(* IEC 61131-3 sources: SRCI/RobotLibrary/Library/POUs/AdvancedMove/MC_MoveLinearOffset, 1 file *)

(* ---- MC_MoveLinearOffsetFB.st ---- *)
/// Move the TCP relative to a reference cartesian position (linear interpolation)
FUNCTION_BLOCK MC_MoveLinearOffsetFB EXTENDS RobotLibraryBaseExecuteFB
// -------------------------------------------------------------------------
//  SRCI Robot Library
// -------------------------------------------------------------------------
//
//  Object:      MoveLinearOffsetFB
//  Author:      Thorsten Brach
//  Date:        2024-06-01
//
//  Description:
//
//
//  Copyright:
//    (C) 2024 Thorsten Brach. All rights reserved
//             Licensed under the LGPL-3.0 license.
//
//  Disclaimer:
//    This project is provided without any guarantee and can be used for
//    private and commercial purposes. Any use is at the user’s
//    own risk and responsibility.
//
// -------------------------------------------------------------------------
VAR_INPUT
  /// Parameter which determines the behavior towards the previously sent and still active or buffered commands
  AbortingMode       : AbortingMode;
  /// Defines the target sequence in which the command will be executed
  SequenceFlag       : SequenceFlag;
  /// command parameter
  ParCmd             : MoveLinearOffsetParCmd;
END_VAR

VAR_OUTPUT
  /// Command is transferred and confirmed by the RC
  CommandBuffered    : BOOL;
  /// The command takes control of the motion of the according axis group
  Active             : BOOL;
  /// The command was aborted by another command.
  CommandAborted     : BOOL;
  /// TRUE, while command is interrupted during execution and can be continued
  CommandInterrupted : BOOL;
  /// command outputs
  OutCmd             : MoveLinearOffsetOutCmd;
END_VAR

VAR
  /// internal copy of command parameter
 _parCmd             : MoveLinearOffsetParCmd;
  /// command data to send
 _command            : MoveLinearOffsetSendData;
  /// response data received
 _response           : MoveLinearOffsetRecvData;
END_VAR

  SUPER^(AxesGroup := AxesGroup);

END_FUNCTION_BLOCK

METHOD INTERNAL CheckAddParameter : BOOL
VAR_INPUT
  /// Payload pointer
  PayloadPtr : UDINT;
END_VAR
VAR
  /// Payload as byte array
  Payload    : ARRAY [1..SIZEOF(_command)] OF BYTE;
  /// Null Byte array
  Null       : ARRAY [1..SIZEOF(_command)] OF BYTE;
  /// Data length to compare
  DataLen    : UDINT;
END_VAR

  // Payload pointer must be decreased by one byte, because ADR(Payload) is already one byte !
  PayloadPtr := LIMIT (0, PayloadPtr - 1, SIZEOF(Payload) -1);
  // Convert command struct to payload array
  SysDepMemCpy( pDest := ADR(Payload), pSrc := ADR(_command), DataLen := SIZEOF(_command));
  // Calculate the data length to compare - at least one byte must be compared !
  DataLen := LIMIT(1, SIZEOF(Payload) - PayloadPtr, SIZEOF(Payload));
  // Compare Payload-Array with Null-Byte-Array
  CheckAddParameter := SysDepMemCmp( pData1 := ADR(Payload) + PayloadPtr , pData2 := ADR(Null), DataLen := DataLen) <>  RobotLibraryConstants.OK ;

END_METHOD

METHOD PROTECTED CheckFunctionSupported : BOOL
VAR_IN_OUT
  /// Robot assignment of function
  AxesGroup : AxesGroup;
END_VAR

  CheckFunctionSupported := AxesGroup.State.RobotData.RCSupportedFunctions.MoveLinearOffset;

  IF ( NOT CheckFunctionSupported )
  THEN
    // call base implementation for set error and create log entry
    SUPER^.CheckFunctionSupported(AxesGroup := AxesGroup);
  END_IF

END_METHOD

METHOD PROTECTED CheckParameterChanged : BOOL
VAR_IN_OUT
  /// Robot assignment of function
  AxesGroup    : AxesGroup;
END_VAR

  // Check ParCmd Size is > 0, because MemCmp does not work correctly with size = 0
  IF (SIZEOF(ParCmd) = 0) OR (_stepCmd = 0)
  THEN
    RETURN;
  END_IF

  // compare memory
  _parameterChanged := ( SysDepMemCmp(pData1 := ADR(ParCmd), pData2 := ADR(_parCmd), DataLen := SIZEOF(ParCmd)) <> RobotLibraryConstants.OK );

  // check parameter valid ?
  _parameterValid   := CheckParameterValid( AxesGroup := AxesGroup );

  IF ((  _parameterChanged        )  AND
      (  _parameterValid          )) OR
      (  _parameterUpdateInternal )
  THEN
    // reset internal flag for send parameter update
   _parameterUpdateInternal := FALSE;
    // update internal copy of parameters
   _parCmd := ParCmd;
    // inc parameter sequence
   _command.ParSeq := _command.ParSeq + 1;
    // update command data
    CommandData := CreateCommandPayload(AxesGroup := AxesGroup); // ( Access via reference to rCommandFB in ACR )
    // notify active command register
    AxesGroup.Acyclic.ActiveCommandRegister.NotifyParameterChanged := _uniqueID;
  END_IF

END_METHOD

METHOD PROTECTED CheckParameterValid : BOOL
VAR_IN_OUT
  /// Robot assignment of function
  AxesGroup : AxesGroup;
END_VAR
VAR
  /// internal index for loops
 _idx : DINT;
END_VAR

  CheckParameterValid := TRUE;

  // Check AbortingMode valid ?
  IF (( AbortingMode <> AbortingModeEnum.BUFFER ) AND
      ( AbortingMode <> AbortingModeEnum.ABORT  ))
  THEN
    // Parameter not valid
    CheckParameterValid := FALSE;
    // Set error
    ErrorID := RobotLibraryErrorIdEnum.ERR_ABORTINGMODE_INVALID;
    // Create log entry
    CreateLogMessagePara1 ( Timestamp   := AxesGroup.State.SystemTime,
                            MessageType := MessageType.CMD,
                            Severity    := Severity.ERROR,
                            MessageCode := ErrorID,
                            MessageText := 'Invalid Parameter AbortingMode = {1}',
                            Para1       := ABORTING_MODE_TO_STRING(AbortingMode));
    RETURN;
  END_IF

  // Check SequenceFlag valid ?
  IF (( SequenceFlag <> SequenceFlagEnum.PRIMARY_SEQUENCE   ) AND
      ( SequenceFlag <> SequenceFlagEnum.SECONDARY_SEQUENCE ))
  THEN
    // Parameter not valid
    CheckParameterValid := FALSE;
    // Set error
    ErrorID := RobotLibraryErrorIdEnum.ERR_SEQFLAG_NOT_ALLOWED;
    // Create log entry
    CreateLogMessagePara1 ( Timestamp   := AxesGroup.State.SystemTime,
                            MessageType := MessageType.CMD,
                            Severity    := Severity.ERROR,
                            MessageCode := ErrorID,
                            MessageText := 'Invalid Parameter SequenceFlag = {1}',
                            Para1       := SEQUENCE_FLAG_TO_STRING(SequenceFlag));
    RETURN;
  END_IF

  // Check ParCmd.ReferencePosition.X valid ?
  IF ( SysDepIsValidReal(ParCmd.ReferencePosition.X) = FALSE )
  THEN
    // Parameter not valid
    CheckParameterValid := FALSE;
    // Set error
    ErrorID := RobotLibraryErrorIdEnum.ERR_INVALID_PAR_CMD;

    // Create log entry
    CreateLogMessagePara1 ( Timestamp   := AxesGroup.State.SystemTime,
                            MessageType := MessageType.CMD,
                            Severity    := Severity.ERROR,
                            MessageCode := ErrorID,
                            MessageText := 'Invalid Parameter ParCmd.ReferencePosition.X = {1}',
                            Para1       := VALID_REAL_TO_STRING(ParCmd.ReferencePosition.X));
    RETURN;
  END_IF

  // Check ParCmd.ReferencePosition.Y valid ?
  IF ( SysDepIsValidReal(ParCmd.ReferencePosition.Y) = FALSE )
  THEN
    // Parameter not valid
    CheckParameterValid := FALSE;
    // Set error
    ErrorID := RobotLibraryErrorIdEnum.ERR_INVALID_PAR_CMD;

    // Create log entry
    CreateLogMessagePara1 ( Timestamp   := AxesGroup.State.SystemTime,
                            MessageType := MessageType.CMD,
                            Severity    := Severity.ERROR,
                            MessageCode := ErrorID,
                            MessageText := 'Invalid Parameter ParCmd.ReferencePosition.Y = {1}',
                            Para1       := VALID_REAL_TO_STRING(ParCmd.ReferencePosition.Y));
    RETURN;
  END_IF

  // Check ParCmd.ReferencePosition.Z valid ?
  IF ( SysDepIsValidReal(ParCmd.ReferencePosition.Z) = FALSE )
  THEN
    // Parameter not valid
    CheckParameterValid := FALSE;
    // Set error
    ErrorID := RobotLibraryErrorIdEnum.ERR_INVALID_PAR_CMD;

    // Create log entry
    CreateLogMessagePara1 ( Timestamp   := AxesGroup.State.SystemTime,
                            MessageType := MessageType.CMD,
                            Severity    := Severity.ERROR,
                            MessageCode := ErrorID,
                            MessageText := 'Invalid Parameter ParCmd.ReferencePosition.Z = {1}',
                            Para1       := VALID_REAL_TO_STRING(ParCmd.ReferencePosition.Z));
    RETURN;
  END_IF

  // Check ParCmd.ReferencePosition.Rx valid ?
  IF ( SysDepIsValidReal(ParCmd.ReferencePosition.Rx) = FALSE )
  THEN
    // Parameter not valid
    CheckParameterValid := FALSE;
    // Set error
    ErrorID := RobotLibraryErrorIdEnum.ERR_INVALID_PAR_CMD;

    // Create log entry
    CreateLogMessagePara1 ( Timestamp   := AxesGroup.State.SystemTime,
                            MessageType := MessageType.CMD,
                            Severity    := Severity.ERROR,
                            MessageCode := ErrorID,
                            MessageText := 'Invalid Parameter ParCmd.ReferencePosition.Rx = {1}',
                            Para1       := VALID_REAL_TO_STRING(ParCmd.ReferencePosition.Rx));
    RETURN;
  END_IF

  // Check ParCmd.ReferencePosition.Ry valid ?
  IF ( SysDepIsValidReal(ParCmd.ReferencePosition.Ry) = FALSE )
  THEN
    // Parameter not valid
    CheckParameterValid := FALSE;
    // Set error
    ErrorID := RobotLibraryErrorIdEnum.ERR_INVALID_PAR_CMD;

    // Create log entry
    CreateLogMessagePara1 ( Timestamp   := AxesGroup.State.SystemTime,
                            MessageType := MessageType.CMD,
                            Severity    := Severity.ERROR,
                            MessageCode := ErrorID,
                            MessageText := 'Invalid Parameter ParCmd.ReferencePosition.Ry = {1}',
                            Para1       := VALID_REAL_TO_STRING(ParCmd.ReferencePosition.Ry));
    RETURN;
  END_IF

  // Check ParCmd.ReferencePosition.Rz valid ?
  IF ( SysDepIsValidReal(ParCmd.ReferencePosition.Rz) = FALSE )
  THEN
    // Parameter not valid
    CheckParameterValid := FALSE;
    // Set error
    ErrorID := RobotLibraryErrorIdEnum.ERR_INVALID_PAR_CMD;

    // Create log entry
    CreateLogMessagePara1 ( Timestamp   := AxesGroup.State.SystemTime,
                            MessageType := MessageType.CMD,
                            Severity    := Severity.ERROR,
                            MessageCode := ErrorID,
                            MessageText := 'Invalid Parameter ParCmd.ReferencePosition.Rz = {1}',
                            Para1       := VALID_REAL_TO_STRING(ParCmd.ReferencePosition.Rz));
    RETURN;
  END_IF

  // Check ParCmd.ReferencePosition.E1 valid ?
  IF ( SysDepIsValidReal(ParCmd.ReferencePosition.E1) = FALSE )
  THEN
    // Parameter not valid
    CheckParameterValid := FALSE;
    // Set error
    ErrorID := RobotLibraryErrorIdEnum.ERR_INVALID_PAR_CMD;

    // Create log entry
    CreateLogMessagePara1 ( Timestamp   := AxesGroup.State.SystemTime,
                            MessageType := MessageType.CMD,
                            Severity    := Severity.ERROR,
                            MessageCode := ErrorID,
                            MessageText := 'Invalid Parameter ParCmd.ReferencePosition.E1 = {1}',
                            Para1       := VALID_REAL_TO_STRING(ParCmd.ReferencePosition.E1));
    RETURN;
  END_IF

  // Check ParCmd.ReferencePosition.E2 valid ?
  IF ( SysDepIsValidReal(ParCmd.ReferencePosition.E2) = FALSE )
  THEN
    // Parameter not valid
    CheckParameterValid := FALSE;
    // Set error
    ErrorID := RobotLibraryErrorIdEnum.ERR_INVALID_PAR_CMD;

    // Create log entry
    CreateLogMessagePara1 ( Timestamp   := AxesGroup.State.SystemTime,
                            MessageType := MessageType.CMD,
                            Severity    := Severity.ERROR,
                            MessageCode := ErrorID,
                            MessageText := 'Invalid Parameter ParCmd.ReferencePosition.E2 = {1}',
                            Para1       := VALID_REAL_TO_STRING(ParCmd.ReferencePosition.E2));
    RETURN;
  END_IF

  // Check ParCmd.ReferencePosition.E3 valid ?
  IF ( SysDepIsValidReal(ParCmd.ReferencePosition.E3) = FALSE )
  THEN
    // Parameter not valid
    CheckParameterValid := FALSE;
    // Set error
    ErrorID := RobotLibraryErrorIdEnum.ERR_INVALID_PAR_CMD;

    // Create log entry
    CreateLogMessagePara1 ( Timestamp   := AxesGroup.State.SystemTime,
                            MessageType := MessageType.CMD,
                            Severity    := Severity.ERROR,
                            MessageCode := ErrorID,
                            MessageText := 'Invalid Parameter ParCmd.ReferencePosition.E3 = {1}',
                            Para1       := VALID_REAL_TO_STRING(ParCmd.ReferencePosition.E3));
    RETURN;
  END_IF

  // Check ParCmd.ReferencePosition.E4 valid ?
  IF ( SysDepIsValidReal(ParCmd.ReferencePosition.E4) = FALSE )
  THEN
    // Parameter not valid
    CheckParameterValid := FALSE;
    // Set error
    ErrorID := RobotLibraryErrorIdEnum.ERR_INVALID_PAR_CMD;

    // Create log entry
    CreateLogMessagePara1 ( Timestamp   := AxesGroup.State.SystemTime,
                            MessageType := MessageType.CMD,
                            Severity    := Severity.ERROR,
                            MessageCode := ErrorID,
                            MessageText := 'Invalid Parameter ParCmd.ReferencePosition.E4 = {1}',
                            Para1       := VALID_REAL_TO_STRING(ParCmd.ReferencePosition.E4));
    RETURN;
  END_IF

  // Check ParCmd.ReferencePosition.E5 valid ?
  IF ( SysDepIsValidReal(ParCmd.ReferencePosition.E5) = FALSE )
  THEN
    // Parameter not valid
    CheckParameterValid := FALSE;
    // Set error
    ErrorID := RobotLibraryErrorIdEnum.ERR_INVALID_PAR_CMD;

    // Create log entry
    CreateLogMessagePara1 ( Timestamp   := AxesGroup.State.SystemTime,
                            MessageType := MessageType.CMD,
                            Severity    := Severity.ERROR,
                            MessageCode := ErrorID,
                            MessageText := 'Invalid Parameter ParCmd.ReferencePosition.E5 = {1}',
                            Para1       := VALID_REAL_TO_STRING(ParCmd.ReferencePosition.E5));
    RETURN;
  END_IF

  // Check ParCmd.ReferencePosition.E6 valid ?
  IF ( SysDepIsValidReal(ParCmd.ReferencePosition.E6) = FALSE )
  THEN
    // Parameter not valid
    CheckParameterValid := FALSE;
    // Set error
    ErrorID := RobotLibraryErrorIdEnum.ERR_INVALID_PAR_CMD;

    // Create log entry
    CreateLogMessagePara1 ( Timestamp   := AxesGroup.State.SystemTime,
                            MessageType := MessageType.CMD,
                            Severity    := Severity.ERROR,
                            MessageCode := ErrorID,
                            MessageText := 'Invalid Parameter ParCmd.ReferencePosition.E6 = {1}',
                            Para1       := VALID_REAL_TO_STRING(ParCmd.ReferencePosition.E6));
    RETURN;
  END_IF

  // Check ParCmd.ReferencePosition.Config.Shoulder valid ?
  IF (( ParCmd.ReferencePosition.Config.Shoulder <> ArmConfigShoulder.USE_CONFIG ) AND
      ( ParCmd.ReferencePosition.Config.Shoulder <> ArmConfigShoulder.SAME       ) AND
      ( ParCmd.ReferencePosition.Config.Shoulder <> ArmConfigShoulder.FREE       ) AND
      ( ParCmd.ReferencePosition.Config.Shoulder <> ArmConfigShoulder.BACK       ) AND
      ( ParCmd.ReferencePosition.Config.Shoulder <> ArmConfigShoulder.FRONT      ))
  THEN
    // Parameter not valid
    CheckParameterValid := FALSE;
    // Set error
    ErrorID := RobotLibraryErrorIdEnum.ERR_CONFIGMODE_SHOULDER_INVALID;
    // Create log entry
    CreateLogMessagePara1 ( Timestamp   := AxesGroup.State.SystemTime,
                            MessageType := MessageType.CMD,
                            Severity    := Severity.ERROR,
                            MessageCode := ErrorID,
                            MessageText := 'Invalid Parameter ParCmd.ReferencePosition.Config.Shoulder = {1}',
                            Para1       :=  ARM_CONFIG_SHOULDER_TO_STRING(ParCmd.ReferencePosition.Config.Shoulder));
    RETURN;
  END_IF

  // Check ParCmd.ReferencePosition.Config.Elbow valid ?
  IF (( ParCmd.ReferencePosition.Config.Elbow <> ArmConfigElbow.USE_CONFIG ) AND
      ( ParCmd.ReferencePosition.Config.Elbow <> ArmConfigElbow.SAME       ) AND
      ( ParCmd.ReferencePosition.Config.Elbow <> ArmConfigElbow.FREE       ) AND
      ( ParCmd.ReferencePosition.Config.Elbow <> ArmConfigElbow.DOWN       ) AND
      ( ParCmd.ReferencePosition.Config.Elbow <> ArmConfigElbow.UP         ))
  THEN
    // Parameter not valid
    CheckParameterValid := FALSE;
    // Set error
    ErrorID := RobotLibraryErrorIdEnum.ERR_CONFIGMODE_ELBOW_INVALID;
    // Create log entry
    CreateLogMessagePara1 ( Timestamp   := AxesGroup.State.SystemTime,
                            MessageType := MessageType.CMD,
                            Severity    := Severity.ERROR,
                            MessageCode := ErrorID,
                            MessageText := 'Invalid Parameter ParCmd.ReferencePosition.Config.Elbow = {1}',
                            Para1       :=  ARM_CONFIG_ELBOW_TO_STRING(ParCmd.ReferencePosition.Config.Elbow));
    RETURN;
  END_IF

  // Check ParCmd.ReferencePosition.Config.Wrist valid ?
  IF (( ParCmd.ReferencePosition.Config.Wrist <> ArmConfigWrist.USE_CONFIG ) AND
      ( ParCmd.ReferencePosition.Config.Wrist <> ArmConfigWrist.SAME       ) AND
      ( ParCmd.ReferencePosition.Config.Wrist <> ArmConfigWrist.FREE       ) AND
      ( ParCmd.ReferencePosition.Config.Wrist <> ArmConfigWrist.FLIP       ) AND
      ( ParCmd.ReferencePosition.Config.Wrist <> ArmConfigWrist.NON_FLIP   ))
  THEN
    // Parameter not valid
    CheckParameterValid := FALSE;
    // Set error
    ErrorID := RobotLibraryErrorIdEnum.ERR_CONFIGMODE_WRIST_INVALID;
    // Create log entry
    CreateLogMessagePara1 ( Timestamp   := AxesGroup.State.SystemTime,
                            MessageType := MessageType.CMD,
                            Severity    := Severity.ERROR,
                            MessageCode := ErrorID,
                            MessageText := 'Invalid Parameter ParCmd.ReferencePosition.Config.Wrist = {1}',
                            Para1       :=  ARM_CONFIG_WRIST_TO_STRING(ParCmd.ReferencePosition.Config.Wrist));
    RETURN;
  END_IF

  // Check ParCmd.Offset.X valid ?
  IF ( SysDepIsValidReal(ParCmd.Offset.X) = FALSE )
  THEN
    // Parameter not valid
    CheckParameterValid := FALSE;
    // Set error
    ErrorID := RobotLibraryErrorIdEnum.ERR_INVALID_PAR_CMD;

    // Create log entry
    CreateLogMessagePara1 ( Timestamp   := AxesGroup.State.SystemTime,
                            MessageType := MessageType.CMD,
                            Severity    := Severity.ERROR,
                            MessageCode := ErrorID,
                            MessageText := 'Invalid Parameter ParCmd.Offset.X = {1}',
                            Para1       := VALID_REAL_TO_STRING(ParCmd.Offset.X));
    RETURN;
  END_IF

  // Check ParCmd.Offset.Y valid ?
  IF ( SysDepIsValidReal(ParCmd.Offset.Y) = FALSE )
  THEN
    // Parameter not valid
    CheckParameterValid := FALSE;
    // Set error
    ErrorID := RobotLibraryErrorIdEnum.ERR_INVALID_PAR_CMD;

    // Create log entry
    CreateLogMessagePara1 ( Timestamp   := AxesGroup.State.SystemTime,
                            MessageType := MessageType.CMD,
                            Severity    := Severity.ERROR,
                            MessageCode := ErrorID,
                            MessageText := 'Invalid Parameter ParCmd.Offset.Y = {1}',
                            Para1       := VALID_REAL_TO_STRING(ParCmd.Offset.Y));
    RETURN;
  END_IF

  // Check ParCmd.Offset.Z valid ?
  IF ( SysDepIsValidReal(ParCmd.Offset.Z) = FALSE )
  THEN
    // Parameter not valid
    CheckParameterValid := FALSE;
    // Set error
    ErrorID := RobotLibraryErrorIdEnum.ERR_INVALID_PAR_CMD;

    // Create log entry
    CreateLogMessagePara1 ( Timestamp   := AxesGroup.State.SystemTime,
                            MessageType := MessageType.CMD,
                            Severity    := Severity.ERROR,
                            MessageCode := ErrorID,
                            MessageText := 'Invalid Parameter ParCmd.Offset.Z = {1}',
                            Para1       := VALID_REAL_TO_STRING(ParCmd.Offset.Z));
    RETURN;
  END_IF

  // Check ParCmd.Offset.Rx valid ?
  IF ( SysDepIsValidReal(ParCmd.Offset.Rx) = FALSE )
  THEN
    // Parameter not valid
    CheckParameterValid := FALSE;
    // Set error
    ErrorID := RobotLibraryErrorIdEnum.ERR_INVALID_PAR_CMD;

    // Create log entry
    CreateLogMessagePara1 ( Timestamp   := AxesGroup.State.SystemTime,
                            MessageType := MessageType.CMD,
                            Severity    := Severity.ERROR,
                            MessageCode := ErrorID,
                            MessageText := 'Invalid Parameter ParCmd.Offset.Rx = {1}',
                            Para1       := VALID_REAL_TO_STRING(ParCmd.Offset.Rx));
    RETURN;
  END_IF

  // Check ParCmd.Offset.Ry valid ?
  IF ( SysDepIsValidReal(ParCmd.Offset.Ry) = FALSE )
  THEN
    // Parameter not valid
    CheckParameterValid := FALSE;
    // Set error
    ErrorID := RobotLibraryErrorIdEnum.ERR_INVALID_PAR_CMD;

    // Create log entry
    CreateLogMessagePara1 ( Timestamp   := AxesGroup.State.SystemTime,
                            MessageType := MessageType.CMD,
                            Severity    := Severity.ERROR,
                            MessageCode := ErrorID,
                            MessageText := 'Invalid Parameter ParCmd.Offset.Ry = {1}',
                            Para1       := VALID_REAL_TO_STRING(ParCmd.Offset.Ry));
    RETURN;
  END_IF

  // Check ParCmd.Offset.Rz valid ?
  IF ( SysDepIsValidReal(ParCmd.Offset.Rz) = FALSE )
  THEN
    // Parameter not valid
    CheckParameterValid := FALSE;
    // Set error
    ErrorID := RobotLibraryErrorIdEnum.ERR_INVALID_PAR_CMD;

    // Create log entry
    CreateLogMessagePara1 ( Timestamp   := AxesGroup.State.SystemTime,
                            MessageType := MessageType.CMD,
                            Severity    := Severity.ERROR,
                            MessageCode := ErrorID,
                            MessageText := 'Invalid Parameter ParCmd.Offset.Rz = {1}',
                            Para1       := VALID_REAL_TO_STRING(ParCmd.Offset.Rz));
    RETURN;
  END_IF

  // Check ParCmd.Offset.E1 valid ?
  IF ( SysDepIsValidReal(ParCmd.Offset.E1) = FALSE )
  THEN
    // Parameter not valid
    CheckParameterValid := FALSE;
    // Set error
    ErrorID := RobotLibraryErrorIdEnum.ERR_INVALID_PAR_CMD;

    // Create log entry
    CreateLogMessagePara1 ( Timestamp   := AxesGroup.State.SystemTime,
                            MessageType := MessageType.CMD,
                            Severity    := Severity.ERROR,
                            MessageCode := ErrorID,
                            MessageText := 'Invalid Parameter ParCmd.Offset.E1 = {1}',
                            Para1       := VALID_REAL_TO_STRING(ParCmd.Offset.E1));
    RETURN;
  END_IF

  // Check ParCmd.Offset.E2 valid ?
  IF ( SysDepIsValidReal(ParCmd.Offset.E2) = FALSE )
  THEN
    // Parameter not valid
    CheckParameterValid := FALSE;
    // Set error
    ErrorID := RobotLibraryErrorIdEnum.ERR_INVALID_PAR_CMD;

    // Create log entry
    CreateLogMessagePara1 ( Timestamp   := AxesGroup.State.SystemTime,
                            MessageType := MessageType.CMD,
                            Severity    := Severity.ERROR,
                            MessageCode := ErrorID,
                            MessageText := 'Invalid Parameter ParCmd.Offset.E2 = {1}',
                            Para1       := VALID_REAL_TO_STRING(ParCmd.Offset.E2));
    RETURN;
  END_IF

  // Check ParCmd.Offset.E3 valid ?
  IF ( SysDepIsValidReal(ParCmd.Offset.E3) = FALSE )
  THEN
    // Parameter not valid
    CheckParameterValid := FALSE;
    // Set error
    ErrorID := RobotLibraryErrorIdEnum.ERR_INVALID_PAR_CMD;

    // Create log entry
    CreateLogMessagePara1 ( Timestamp   := AxesGroup.State.SystemTime,
                            MessageType := MessageType.CMD,
                            Severity    := Severity.ERROR,
                            MessageCode := ErrorID,
                            MessageText := 'Invalid Parameter ParCmd.Offset.E3 = {1}',
                            Para1       := VALID_REAL_TO_STRING(ParCmd.Offset.E3));
    RETURN;
  END_IF

  // Check ParCmd.Offset.E4 valid ?
  IF ( SysDepIsValidReal(ParCmd.Offset.E4) = FALSE )
  THEN
    // Parameter not valid
    CheckParameterValid := FALSE;
    // Set error
    ErrorID := RobotLibraryErrorIdEnum.ERR_INVALID_PAR_CMD;

    // Create log entry
    CreateLogMessagePara1 ( Timestamp   := AxesGroup.State.SystemTime,
                            MessageType := MessageType.CMD,
                            Severity    := Severity.ERROR,
                            MessageCode := ErrorID,
                            MessageText := 'Invalid Parameter ParCmd.Offset.E4 = {1}',
                            Para1       := VALID_REAL_TO_STRING(ParCmd.Offset.E4));
    RETURN;
  END_IF

  // Check ParCmd.Offset.E5 valid ?
  IF ( SysDepIsValidReal(ParCmd.Offset.E5) = FALSE )
  THEN
    // Parameter not valid
    CheckParameterValid := FALSE;
    // Set error
    ErrorID := RobotLibraryErrorIdEnum.ERR_INVALID_PAR_CMD;

    // Create log entry
    CreateLogMessagePara1 ( Timestamp   := AxesGroup.State.SystemTime,
                            MessageType := MessageType.CMD,
                            Severity    := Severity.ERROR,
                            MessageCode := ErrorID,
                            MessageText := 'Invalid Parameter ParCmd.Offset.E5 = {1}',
                            Para1       := VALID_REAL_TO_STRING(ParCmd.Offset.E5));
    RETURN;
  END_IF

  // Check ParCmd.Offset.E6 valid ?
  IF ( SysDepIsValidReal(ParCmd.Offset.E6) = FALSE )
  THEN
    // Parameter not valid
    CheckParameterValid := FALSE;
    // Set error
    ErrorID := RobotLibraryErrorIdEnum.ERR_INVALID_PAR_CMD;

    // Create log entry
    CreateLogMessagePara1 ( Timestamp   := AxesGroup.State.SystemTime,
                            MessageType := MessageType.CMD,
                            Severity    := Severity.ERROR,
                            MessageCode := ErrorID,
                            MessageText := 'Invalid Parameter ParCmd.Offset.E6 = {1}',
                            Para1       := VALID_REAL_TO_STRING(ParCmd.Offset.E6));
    RETURN;
  END_IF

  // Check ParCmd.Offset.Config.Shoulder valid ?
  IF (( ParCmd.Offset.Config.Shoulder <> ArmConfigShoulder.USE_CONFIG ) AND
      ( ParCmd.Offset.Config.Shoulder <> ArmConfigShoulder.SAME       ) AND
      ( ParCmd.Offset.Config.Shoulder <> ArmConfigShoulder.FREE       ) AND
      ( ParCmd.Offset.Config.Shoulder <> ArmConfigShoulder.BACK       ) AND
      ( ParCmd.Offset.Config.Shoulder <> ArmConfigShoulder.FRONT      ))
  THEN
    // Parameter not valid
    CheckParameterValid := FALSE;
    // Set error
    ErrorID := RobotLibraryErrorIdEnum.ERR_CONFIGMODE_SHOULDER_INVALID;
    // Create log entry
    CreateLogMessagePara1 ( Timestamp   := AxesGroup.State.SystemTime,
                            MessageType := MessageType.CMD,
                            Severity    := Severity.ERROR,
                            MessageCode := ErrorID,
                            MessageText := 'Invalid Parameter ParCmd.Offset.Config.Shoulder = {1}',
                            Para1       :=  ARM_CONFIG_SHOULDER_TO_STRING(ParCmd.Offset.Config.Shoulder));
    RETURN;
  END_IF

  // Check ParCmd.Offset.Config.Elbow valid ?
  IF (( ParCmd.Offset.Config.Elbow <> ArmConfigElbow.USE_CONFIG ) AND
      ( ParCmd.Offset.Config.Elbow <> ArmConfigElbow.SAME       ) AND
      ( ParCmd.Offset.Config.Elbow <> ArmConfigElbow.FREE       ) AND
      ( ParCmd.Offset.Config.Elbow <> ArmConfigElbow.DOWN       ) AND
      ( ParCmd.Offset.Config.Elbow <> ArmConfigElbow.UP         ))
  THEN
    // Parameter not valid
    CheckParameterValid := FALSE;
    // Set error
    ErrorID := RobotLibraryErrorIdEnum.ERR_CONFIGMODE_ELBOW_INVALID;
    // Create log entry
    CreateLogMessagePara1 ( Timestamp   := AxesGroup.State.SystemTime,
                            MessageType := MessageType.CMD,
                            Severity    := Severity.ERROR,
                            MessageCode := ErrorID,
                            MessageText := 'Invalid Parameter ParCmd.Offset.Config.Elbow = {1}',
                            Para1       :=  ARM_CONFIG_ELBOW_TO_STRING(ParCmd.Offset.Config.Elbow));
    RETURN;
  END_IF

  // Check ParCmd.Offset.Config.Wrist valid ?
  IF (( ParCmd.Offset.Config.Wrist <> ArmConfigWrist.USE_CONFIG ) AND
      ( ParCmd.Offset.Config.Wrist <> ArmConfigWrist.SAME       ) AND
      ( ParCmd.Offset.Config.Wrist <> ArmConfigWrist.FREE       ) AND
      ( ParCmd.Offset.Config.Wrist <> ArmConfigWrist.FLIP       ) AND
      ( ParCmd.Offset.Config.Wrist <> ArmConfigWrist.NON_FLIP   ))
  THEN
    // Parameter not valid
    CheckParameterValid := FALSE;
    // Set error
    ErrorID := RobotLibraryErrorIdEnum.ERR_CONFIGMODE_WRIST_INVALID;
    // Create log entry
    CreateLogMessagePara1 ( Timestamp   := AxesGroup.State.SystemTime,
                            MessageType := MessageType.CMD,
                            Severity    := Severity.ERROR,
                            MessageCode := ErrorID,
                            MessageText := 'Invalid Parameter ParCmd.Offset.Config.Wrist = {1}',
                            Para1       :=  ARM_CONFIG_WRIST_TO_STRING(ParCmd.Offset.Config.Wrist));
    RETURN;
  END_IF

  // Check ParCmd.ReferenceType valid ?
  IF (( ParCmd.ReferenceType <> ReferenceType.TOOL  ) AND
      ( ParCmd.ReferenceType <> ReferenceType.FRAME ))
  THEN
    // Parameter not valid
    CheckParameterValid := FALSE;
    // Set error
    ErrorID := RobotLibraryErrorIdEnum.ERR_INVALID_PAR_CMD;
    // Create log entry
    CreateLogMessagePara1 ( Timestamp   := AxesGroup.State.SystemTime,
                            MessageType := MessageType.CMD,
                            Severity    := Severity.ERROR,
                            MessageCode := ErrorID,
                            MessageText := 'Invalid Parameter ParCmd.ReferenceType = {1}',
                            Para1       := REFERENCE_TYPE_TO_STRING(ParCmd.ReferenceType));
    RETURN;
  END_IF

  // Check ParCmd.VelocityRate valid ?
  IF  (( SysDepIsValidReal(ParCmd.VelocityRate) = FALSE )  OR
      ((                   ParCmd.VelocityRate  <     0 )  AND
       (                   ParCmd.VelocityRate <>    -1 )) OR
       (                   ParCmd.VelocityRate  >   100 ))
  THEN
    // Parameter not valid
    CheckParameterValid := FALSE;
    // Set error
    ErrorID := RobotLibraryErrorIdEnum.ERR_VELOCITY_INVALID;
    // Create log entry
    CreateLogMessagePara1 ( Timestamp   := AxesGroup.State.SystemTime,
                            MessageType := MessageType.CMD,
                            Severity    := Severity.ERROR,
                            MessageCode := ErrorID,
                            MessageText := 'Invalid Parameter ParCmd.VelocityRate = {1}',
                            Para1       := VALID_REAL_TO_STRING(ParCmd.VelocityRate));
    RETURN;
  END_IF

  // Check ParCmd.AccelerationRate valid ?
  IF  (( SysDepIsValidReal(ParCmd.AccelerationRate) = FALSE )  OR
      ((                   ParCmd.AccelerationRate  <     0 )  AND
       (                   ParCmd.AccelerationRate <>    -1 )) OR
       (                   ParCmd.AccelerationRate  >   100 ))
  THEN
    // Parameter not valid
    CheckParameterValid := FALSE;
    // Set error
    ErrorID := RobotLibraryErrorIdEnum.ERR_ACCELERATION_INVALID;
    // Create log entry
    CreateLogMessagePara1 ( Timestamp   := AxesGroup.State.SystemTime,
                            MessageType := MessageType.CMD,
                            Severity    := Severity.ERROR,
                            MessageCode := ErrorID,
                            MessageText := 'Invalid Parameter ParCmd.AccelerationRate = {1}',
                            Para1       := VALID_REAL_TO_STRING(ParCmd.AccelerationRate));
    RETURN;
  END_IF

  // Check ParCmd.DecelerationRate valid ?
  IF  (( SysDepIsValidReal(ParCmd.DecelerationRate) = FALSE )  OR
      ((                   ParCmd.DecelerationRate  <     0 )  AND
       (                   ParCmd.DecelerationRate <>    -1 )) OR
       (                   ParCmd.DecelerationRate  >   100 ))
  THEN
    // Parameter not valid
    CheckParameterValid := FALSE;
    // Set error
    ErrorID := RobotLibraryErrorIdEnum.ERR_DECELERATION_INVALID;
    // Create log entry
    CreateLogMessagePara1 ( Timestamp   := AxesGroup.State.SystemTime,
                            MessageType := MessageType.CMD,
                            Severity    := Severity.ERROR,
                            MessageCode := ErrorID,
                            MessageText := 'Invalid Parameter ParCmd.DecelerationRate = {1}',
                            Para1       := VALID_REAL_TO_STRING(ParCmd.DecelerationRate));
    RETURN;
  END_IF

  // Check ParCmd.JerkRate valid ?
  IF  (( SysDepIsValidReal(ParCmd.JerkRate) = FALSE )  OR
      ((                   ParCmd.JerkRate  <     0 )  AND
       (                   ParCmd.JerkRate <>    -1 )) OR
       (                   ParCmd.JerkRate  >   100 ))
  THEN
    // Parameter not valid
    CheckParameterValid := FALSE;
    // Set error
    ErrorID := RobotLibraryErrorIdEnum.ERR_JERK_INVALID;
    // Create log entry
    CreateLogMessagePara1 ( Timestamp   := AxesGroup.State.SystemTime,
                            MessageType := MessageType.CMD,
                            Severity    := Severity.ERROR,
                            MessageCode := ErrorID,
                            MessageText := 'Invalid Parameter ParCmd.JerkRate = {1}',
                            Para1       := VALID_REAL_TO_STRING(ParCmd.JerkRate));
    RETURN;
  END_IF

  // Check ParCmd.ToolNo valid ?
  IF (( ParCmd.ToolNo <   0                                                ) OR
      ( ParCmd.ToolNo > 254                                                ) OR
      ( ParCmd.ToolNo > AxesGroup.State.ConfigurationData.HighestToolIndex ) OR
      ( ParCmd.ToolNo > RobotLibraryParameter.TOOL_MAX -1                  ))
  THEN
    // Parameter not valid
    CheckParameterValid := FALSE;

    // Check ToolNo available on RC ?
    IF ( ParCmd.ToolNo > AxesGroup.State.ConfigurationData.HighestToolIndex )
    THEN
      ErrorID := RobotLibraryErrorIdEnum.ERR_TOOLNO_UNAVAILABLE;
    ELSE
      ErrorID := RobotLibraryErrorIdEnum.ERR_TOOLNO_RANGE;
  	END_IF

    // Create log entry
    CreateLogMessagePara1 ( Timestamp   := AxesGroup.State.SystemTime,
                            MessageType := MessageType.CMD,
                            Severity    := Severity.ERROR,
                            MessageCode := ErrorID,
                            MessageText := 'Invalid Parameter ParCmd.ToolNo = {1}',
                            Para1       := USINT_TO_STRING(ParCmd.ToolNo));
    RETURN;
  END_IF

  // Check ParCmd.FrameNo valid ?
  IF (( ParCmd.FrameNo <   0                                                 ) OR
      ( ParCmd.FrameNo > 254                                                 ) OR
      ( ParCmd.FrameNo > AxesGroup.State.ConfigurationData.HighestFrameIndex ) OR
      ( ParCmd.FrameNo > RobotLibraryParameter.FRAME_MAX -1                  ))
  THEN
    // Parameter not valid
    CheckParameterValid := FALSE;

    // Check FrameNo available on RC ?
    IF ( ParCmd.FrameNo > AxesGroup.State.ConfigurationData.HighestFrameIndex )
    THEN
      ErrorID := RobotLibraryErrorIdEnum.ERR_FRAMENO_UNAVAILABLE;
    ELSE
      ErrorID := RobotLibraryErrorIdEnum.ERR_FRAMENO_RANGE;
  	END_IF

    // Create log entry
    CreateLogMessagePara1 ( Timestamp   := AxesGroup.State.SystemTime,
                            MessageType := MessageType.CMD,
                            Severity    := Severity.ERROR,
                            MessageCode := ErrorID,
                            MessageText := 'Invalid Parameter ParCmd.FrameNo = {1}',
                            Para1       := USINT_TO_STRING(ParCmd.FrameNo));
    RETURN;
  END_IF

  // Check ParCmd.BlendingMode valid ?
  IF (( ParCmd.BlendingMode <> BlendingMode.EXACT_STOP           ) AND
      ( ParCmd.BlendingMode <> BlendingMode.DEFINED_VELOCITY     ) AND
      ( ParCmd.BlendingMode <> BlendingMode.CORNER_DISTANCE      ) AND
      ( ParCmd.BlendingMode <> BlendingMode.MAX_CORNER_DEVIATION ) AND
      ( ParCmd.BlendingMode <> BlendingMode.CORNER_DISTANCE_2R   ) AND
      ( ParCmd.BlendingMode <> BlendingMode.RAMP_OVERLAP         ) AND
      ( ParCmd.BlendingMode <> BlendingMode.CORNER_DISTANCE_1R   ))
  THEN
    // Parameter not valid
    CheckParameterValid := FALSE;
    // Set error
    ErrorID := RobotLibraryErrorIdEnum.ERR_INVALID_PAR_CMD;
    // Create log entry
    CreateLogMessagePara1 ( Timestamp   := AxesGroup.State.SystemTime,
                            MessageType := MessageType.CMD,
                            Severity    := Severity.ERROR,
                            MessageCode := ErrorID,
                            MessageText := 'Invalid Parameter ParCmd.BlendingMode = {1}',
                            Para1       := BLENDING_MODE_TO_STRING(ParCmd.BlendingMode));
    RETURN;
  END_IF

  FOR _idx := 0 TO 1
  DO
    // Check ParCmd.BlendingParameter valid ?
    IF  ( SysDepIsValidReal(ParCmd.BlendingParameter[_idx]) = FALSE )
    THEN
      // Parameter not valid
      CheckParameterValid := FALSE;
      // Set error
      ErrorID := RobotLibraryErrorIdEnum.ERR_JERK_INVALID;
      // Create log entry
      CreateLogMessagePara2 ( Timestamp   := AxesGroup.State.SystemTime,
                              MessageType := MessageType.CMD,
                              Severity    := Severity.ERROR,
                              MessageCode := ErrorID,
                              MessageText := 'Invalid Parameter ParCmd.BlendingParameter[{2}] = {1}',
                              Para1       := VALID_REAL_TO_STRING(ParCmd.JerkRate),
                              Para2       := DINT_TO_STRING(_idx));
      EXIT;
      RETURN;
    END_IF
  END_FOR

  // Check ParCmd.MoveTime valid ?
  IF  ( ParCmd.MoveTime < T#0S )
  THEN
    // Parameter not valid
    CheckParameterValid := FALSE;
    // Set error
    ErrorID := RobotLibraryErrorIdEnum.ERR_INVALID_PAR_CMD;
    // Create log entry
    CreateLogMessagePara1 ( Timestamp   := AxesGroup.State.SystemTime,
                            MessageType := MessageType.CMD,
                            Severity    := Severity.ERROR,
                            MessageCode := ErrorID,
                            MessageText := 'Invalid Parameter ParCmd.MoveTime = {1}',
                            Para1       := TIME_TO_STRING(ParCmd.MoveTime));
    RETURN;
  END_IF

  // Check ParCmd.OriMode valid ?
  IF (( ParCmd.OriMode <> OriMode.LINEAR_INTERPOLATED ) AND
      ( ParCmd.OriMode <> OriMode.JOINT_INTERPOLATED  ) AND
      ( ParCmd.OriMode <> OriMode.FIX                 ) AND
      ( ParCmd.OriMode <> OriMode.PATH                ))
  THEN
    // Parameter not valid
    CheckParameterValid := FALSE;
    // Set error
    ErrorID := RobotLibraryErrorIdEnum.ERR_INVALID_PAR_CMD;
    // Create log entry
    CreateLogMessagePara1 ( Timestamp   := AxesGroup.State.SystemTime,
                            MessageType := MessageType.CMD,
                            Severity    := Severity.ERROR,
                            MessageCode := ErrorID,
                            MessageText := 'Invalid Parameter ParCmd.OriMode = {1}',
                            Para1       := ORI_MODE_TO_STRING(ParCmd.OriMode));
    RETURN;
  END_IF

  // Check ParCmd.ConfigMode.Shoulder valid ?
  IF (( ParCmd.ConfigMode.Shoulder <> ArmConfigShoulder.USE_CONFIG ) AND
      ( ParCmd.ConfigMode.Shoulder <> ArmConfigShoulder.SAME       ) AND
      ( ParCmd.ConfigMode.Shoulder <> ArmConfigShoulder.FREE       ) AND
      ( ParCmd.ConfigMode.Shoulder <> ArmConfigShoulder.BACK       ) AND
      ( ParCmd.ConfigMode.Shoulder <> ArmConfigShoulder.FRONT      ))
  THEN
    // Parameter not valid
    CheckParameterValid := FALSE;
    // Set error
    ErrorID := RobotLibraryErrorIdEnum.ERR_INVALID_PAR_CMD;
    // Create log entry
    CreateLogMessagePara1 ( Timestamp   := AxesGroup.State.SystemTime,
                            MessageType := MessageType.CMD,
                            Severity    := Severity.ERROR,
                            MessageCode := ErrorID,
                            MessageText := 'Invalid Parameter ParCmd.ConfigMode.Shoulder = {1}',
                            Para1       :=  ARM_CONFIG_SHOULDER_TO_STRING(ParCmd.ConfigMode.Shoulder));
    RETURN;
  END_IF

  // Check ParCmd.ConfigMode.Elbow valid ?
  IF (( ParCmd.ConfigMode.Elbow <> ArmConfigElbow.USE_CONFIG ) AND
      ( ParCmd.ConfigMode.Elbow <> ArmConfigElbow.SAME       ) AND
      ( ParCmd.ConfigMode.Elbow <> ArmConfigElbow.FREE       ) AND
      ( ParCmd.ConfigMode.Elbow <> ArmConfigElbow.DOWN       ) AND
      ( ParCmd.ConfigMode.Elbow <> ArmConfigElbow.UP         ))
  THEN
    // Parameter not valid
    CheckParameterValid := FALSE;
    // Set error
    ErrorID := RobotLibraryErrorIdEnum.ERR_INVALID_PAR_CMD;
    // Create log entry
    CreateLogMessagePara1 ( Timestamp   := AxesGroup.State.SystemTime,
                            MessageType := MessageType.CMD,
                            Severity    := Severity.ERROR,
                            MessageCode := ErrorID,
                            MessageText := 'Invalid Parameter ParCmd.ConfigMode.Elbow = {1}',
                            Para1       :=  ARM_CONFIG_ELBOW_TO_STRING(ParCmd.ConfigMode.Elbow));
    RETURN;
  END_IF

  // Check ParCmd.ConfigMode.Wrist valid ?
  IF (( ParCmd.ConfigMode.Wrist <> ArmConfigWrist.USE_CONFIG ) AND
      ( ParCmd.ConfigMode.Wrist <> ArmConfigWrist.SAME       ) AND
      ( ParCmd.ConfigMode.Wrist <> ArmConfigWrist.FREE       ) AND
      ( ParCmd.ConfigMode.Wrist <> ArmConfigWrist.FLIP       ) AND
      ( ParCmd.ConfigMode.Wrist <> ArmConfigWrist.NON_FLIP   ))
  THEN
    // Parameter not valid
    CheckParameterValid := FALSE;
    // Set error
    ErrorID := RobotLibraryErrorIdEnum.ERR_INVALID_PAR_CMD;
    // Create log entry
    CreateLogMessagePara1 ( Timestamp   := AxesGroup.State.SystemTime,
                            MessageType := MessageType.CMD,
                            Severity    := Severity.ERROR,
                            MessageCode := ErrorID,
                            MessageText := 'Invalid Parameter ParCmd.ConfigMode.Wrist = {1}',
                            Para1       :=  ARM_CONFIG_WRIST_TO_STRING(ParCmd.ConfigMode.Wrist));
    RETURN;
  END_IF

  // Check ParCmd.TurnMode valid ?
  IF (( ParCmd.TurnMode <> TurnMode.USE_TURN_NUMBER ) AND
      ( ParCmd.TurnMode <> TurnMode.SAME            ) AND
      ( ParCmd.TurnMode <> TurnMode.FREE            ))
  THEN
    // Parameter not valid
    CheckParameterValid := FALSE;
    // Set error
    ErrorID := RobotLibraryErrorIdEnum.ERR_INVALID_PAR_CMD;
    // Create log entry
    CreateLogMessagePara1 ( Timestamp   := AxesGroup.State.SystemTime,
                            MessageType := MessageType.CMD,
                            Severity    := Severity.ERROR,
                            MessageCode := ErrorID,
                            MessageText := 'Invalid Parameter ParCmd.TurnMode = {1}',
                            Para1       :=  TURN_MODE_TO_STRING(ParCmd.TurnMode));
    RETURN;
  END_IF

  // Check ParCmd.Manipulation
  // -> no plausibility check for boolean

  FOR _idx := 0 TO 3
  DO
    // Check ParCmd.EmitterID valid ?
    IF  (( ParCmd.EmitterID[_idx] < -127 ) OR
         ( ParCmd.EmitterID[_idx] >  127 ))
    THEN
      // Parameter not valid
      CheckParameterValid := FALSE;
      // Set error
      ErrorID := RobotLibraryErrorIdEnum.ERR_INVALID_PAR_CMD;
      // Create log entry
      CreateLogMessagePara2 ( Timestamp   := AxesGroup.State.SystemTime,
                              MessageType := MessageType.CMD,
                              Severity    := Severity.ERROR,
                              MessageCode := ErrorID,
                              MessageText := 'Invalid Parameter ParCmd.EmitterID[{2}] = {1}',
                              Para1       := SINT_TO_STRING(ParCmd.EmitterID[_idx]),
                              Para2       := DINT_TO_STRING(_idx));
      EXIT;
      RETURN;
    END_IF
  END_FOR

END_METHOD

METHOD INTERNAL CreateCommandPayload : RobotLibraryCommandDataFB
VAR_IN_OUT
  /// Robot assignment of function
  AxesGroup : AxesGroup;
END_VAR
VAR
  /// internal index for loops
 _idx          : DINT;
  /// Parameter count
 _parameterCnt : DINT;
END_VAR
// Table 6-344: Sent CMD payload (PLC to RC) of "MoveLinearOffset"
// --------------------------
// Header
// --------------------------
// Byte 00 : UINT  - Type HB
// Byte 01 :       - Type LB
// Byte 02 : USINT - Reserve | ExecutionMode
// Byte 03 : USINT - ParSeq  | Priority
// --------------------------
// Datablock
// --------------------------
// Byte 04 : SINT  - EmitterID[0];
// Byte 05 : SINT  - EmitterID[1];
// Byte 06 : SINT  - EmitterID[2];
// Byte 07 : SINT  - EmitterID[3];
// Byte 08 : SINT  - ListenerID;
// Byte 09 : BYTE  - Reserved;
// Byte 10 : UINT  - VelocityRate HB;
// Byte 11 :       - VelocityRate LB;
// Byte 12 : UINT  - AccelerationRate HW HB;
// Byte 13 :       - AccelerationRate HW LB;
// Byte 14 : UINT  - DecelerationRate HW HB;
// Byte 15 :       - DecelerationRate HW LB;
// Byte 16 : UINT  - JerkRate HB;
// Byte 17 :       - JerkRate LB;
// Byte 18 : USINT - ToolNo;
// Byte 19 : USINT - FrameNo;
// Byte 20 : USINT - BlendingMode;
// Byte 21 : USINT - OriMode;
// Byte 22 : REAL  - BlendingParameter[0] HW HB;
// Byte 23 :       - BlendingParameter[0] HW LB;
// Byte 24 :       - BlendingParameter[0] LW HB;
// Byte 25 :       - BlendingParameter[0] LW LB;
// Byte 26 : REAL  - BlendingParameter[1] HW HB;
// Byte 27 :       - BlendingParameter[1] HW LB;
// Byte 28 :       - BlendingParameter[1] LW HB;
// Byte 29 :       - BlendingParameter[1] LW LB;
// Byte 30 : REAL  - ReferencePosition.X HW HB;
// Byte 31 :       - ReferencePosition.X HW LB;
// Byte 32 :       - ReferencePosition.X LW HB;
// Byte 33 :       - ReferencePosition.X LW LB;
// Byte 34 : REAL  - ReferencePosition.Y HW HB;
// Byte 35 :       - ReferencePosition.Y HW LB;
// Byte 36 :       - ReferencePosition.Y LW HB;
// Byte 37 :       - ReferencePosition.Y LW LB;
// Byte 38 : REAL  - ReferencePosition.Z HW HB;
// Byte 39 :       - ReferencePosition.Z HW LB;
// Byte 40 :       - ReferencePosition.Z LW HB;
// Byte 41 :       - ReferencePosition.Z LW LB;
// Byte 42 : REAL  - ReferencePosition.RX HW HB;
// Byte 43 :       - ReferencePosition.RX HW LB;
// Byte 44 :       - ReferencePosition.RX LW HB;
// Byte 45 :       - ReferencePosition.RX LW LB;
// Byte 46 : REAL  - ReferencePosition.RY HW HB;
// Byte 47 :       - ReferencePosition.RY HW LB;
// Byte 48 :       - ReferencePosition.RY LW HB;
// Byte 49 :       - ReferencePosition.RY LW LB;
// Byte 50 : REAL  - ReferencePosition.RZ HW HB;
// Byte 51 :       - ReferencePosition.RZ HW LB;
// Byte 52 :       - ReferencePosition.RZ LW HB;
// Byte 53 :       - ReferencePosition.RZ LW LB;
// Byte 54 : BYTE  - - - - - - W E S;
// Byte 55 : BYTE  - Reserved;
// Byte 56 : BYTE  - ReferencePosition.TurnNumber[0];
// Byte 57 : BYTE  - ReferencePosition.TurnNumber[1];
// Byte 58 : BYTE  - ReferencePosition.TurnNumber[2];
// Byte 59 : BYTE  - ReferencePosition.TurnNumber[3];
// Byte 60 : REAL  - ReferencePosition.E1 HW HB;
// Byte 61 :       - ReferencePosition.E1 HW LB;
// Byte 62 :       - ReferencePosition.E1 LW HB;
// Byte 63 :       - ReferencePosition.E1 LW LB;
// Byte 64 : REAL  - Offset.X HW HB;
// Byte 65 :       - Offset.X HW LB;
// Byte 66 :       - Offset.X LW HB;
// Byte 67 :       - Offset.X LW LB;
// Byte 68 : REAL  - Offset.Y HW HB;
// Byte 69 :       - Offset.Y HW LB;
// Byte 70 :       - Offset.Y LW HB;
// Byte 71 :       - Offset.Y LW LB;
// Byte 72 : REAL  - Offset.Z HW HB;
// Byte 73 :       - Offset.Z HW LB;
// Byte 74 :       - Offset.Z LW HB;
// Byte 75 :       - Offset.Z LW LB;
// Byte 76 : REAL  - Offset.RX HW HB;
// Byte 77 :       - Offset.RX HW LB;
// Byte 78 :       - Offset.RX LW HB;
// Byte 79 :       - Offset.RX LW LB;
// Byte 80 : REAL  - Offset.RY HW HB;
// Byte 81 :       - Offset.RY HW LB;
// Byte 82 :       - Offset.RY LW HB;
// Byte 83 :       - Offset.RY LW LB;
// Byte 84 : REAL  - Offset.RZ HW HB;
// Byte 85 :       - Offset.RZ HW LB;
// Byte 86 :       - Offset.RZ LW HB;
// Byte 87 :       - Offset.RZ LW LB;
// Byte 88 : BYTE  - - - - - - W E S;
// Byte 89 : BYTE  - Reserved;
// Byte 90 : BYTE  - Offset.TurnNumber[0];
// Byte 91 : BYTE  - Offset.TurnNumber[1];
// Byte 92 : BYTE  - Offset.TurnNumber[2];
// Byte 93 : BYTE  - Offset.TurnNumber[3];
// Byte 94 : REAL  - Offset.E1 HW HB;
// Byte 95 :       - Offset.E1 HW LB;
// Byte 96 :       - Offset.E1 LW HB;
// Byte 97 :       - Offset.E1 LW LB;
// Byte 98 : BOOL  - Manipulation;
// Byte 99 : BYTE  - Reserved;
// Byte 100: BYTE  - ConfigMode[0];
// Byte 101: BYTE  - ConfigMode[1];
// Byte 102: USINT - ReferenceType;
// Byte 103: USINT - TurnMode;
// Byte 104: UINT  - Time HB;
// Byte 105:       - Time LB;
// Byte 106: REAL  - ReferencePosition.E2 HW HB;
// Byte 107:       - ReferencePosition.E2 HW LB;
// Byte 108:       - ReferencePosition.E2 LW HB;
// Byte 109:       - ReferencePosition.E2 LW LB;
// Byte 110: REAL  - ReferencePosition.E3 HW HB;
// Byte 111:       - ReferencePosition.E3 HW LB;
// Byte 112:       - ReferencePosition.E3 LW HB;
// Byte 113:       - ReferencePosition.E3 LW LB;
// Byte 114: REAL  - ReferencePosition.E4 HW HB;
// Byte 115:       - ReferencePosition.E4 HW LB;
// Byte 116:       - ReferencePosition.E4 LW HB;
// Byte 117:       - ReferencePosition.E4 LW LB;
// Byte 118: REAL  - ReferencePosition.E5 HW HB;
// Byte 119:       - ReferencePosition.E5 HW LB;
// Byte 120:       - ReferencePosition.E5 LW HB;
// Byte 121:       - ReferencePosition.E5 LW LB;
// Byte 122: REAL  - ReferencePosition.E6 HW HB;
// Byte 123:       - ReferencePosition.E6 HW LB;
// Byte 124:       - ReferencePosition.E6 LW HB;
// Byte 125:       - ReferencePosition.E6 LW LB;
// Byte 126: REAL  - Offset.E2 HW HB;
// Byte 127:       - Offset.E2 HW LB;
// Byte 128:       - Offset.E2 LW HB;
// Byte 129:       - Offset.E2 LW LB;
// Byte 130: REAL  - Offset.E3 HW HB;
// Byte 131:       - Offset.E3 HW LB;
// Byte 132:       - Offset.E3 LW HB;
// Byte 133:       - Offset.E3 LW LB;
// Byte 134: REAL  - Offset.E4 HW HB;
// Byte 135:       - Offset.E4 HW LB;
// Byte 136:       - Offset.E4 LW HB;
// Byte 137:       - Offset.E4 LW LB;
// Byte 138: REAL  - Offset.E5 HW HB;
// Byte 139:       - Offset.E5 HW LB;
// Byte 140:       - Offset.E5 LW HB;
// Byte 141:       - Offset.E5 LW LB;
// Byte 142: REAL  - Offset.E6 HW HB;
// Byte 143:       - Offset.E6 HW LB;
// Byte 144:       - Offset.E6 LW HB;
// Byte 145:       - Offset.E6 LW LB;
// --------------------------

  // set command parameter
  _command.CmdTyp            :=  CmdType.MoveLinearOffset;
  _command.ExecMode          :=  ExecMode;
  _command.ParSeq            := _command.ParSeq;
  _command.Priority          :=  Priority;
  _command.EmitterID         := _parCmd.EmitterID;
  _command.ListenerID        := 0;
  _command.Reserve           := 0;
  _command.VelocityRate      := REAL_TO_PERCENT_UINT(_parCmd.VelocityRate     , IsOptional := FALSE);
  _command.AccelerationRate  := REAL_TO_PERCENT_UINT(_parCmd.AccelerationRate , IsOptional := FALSE);
  _command.DecelerationRate  := REAL_TO_PERCENT_UINT(_parCmd.DecelerationRate , IsOptional := TRUE );
  _command.JerkRate          := REAL_TO_PERCENT_UINT(_parCmd.JerkRate         , IsOptional := TRUE );
  _command.ToolNo            := _parCmd.ToolNo;
  _command.FrameNo           := _parCmd.FrameNo;
  _command.BlendingMode      := _parCmd.BlendingMode;
  _command.OriMode           := _parCmd.OriMode;
  _command.BlendingParameter := _parCmd.BlendingParameter;
  _command.ReferencePosition := _parCmd.ReferencePosition;
  _command.Offset            := _parCmd.Offset;
  _command.Manipulation      := _parCmd.Manipulation;
  _command.Reserve2          := 0;
  _command.ConfigMode        :=  ArmConfigParameterToBytes(_parCmd.ConfigMode);
  _command.ReferenceType     := _parCmd.ReferenceType;
  _command.TurnMode          := _parCmd.TurnMode;
  _command.MoveTime          := TIME_TO_UINT(_parCmd.MoveTime);

  // copy command data to header
  _cmdHeader := _command;
  // call base implementation to copy header to payload buffer
  CreateCommandPayload := SUPER^.CreateCommandPayload(AxesGroup := AxesGroup);

  FOR _idx := 0 TO 3
  DO
    // Check parameter must be added ?
    IF ( CheckAddParameter(CreateCommandPayload.PayloadPtr))
    THEN
      // add command.EmitterID[x]
      CreateCommandPayload.AddSint(_command.EmitterID[_idx]);
      // inc parameter counter
     _parameterCnt := _parameterCnt + 1;
    END_IF
  END_FOR

  // Check parameter must be added ?
  IF ( CheckAddParameter(CreateCommandPayload.PayloadPtr))
  THEN
    // add command.ListenerID
    CreateCommandPayload.AddSint(_command.ListenerID);
    // inc parameter counter
   _parameterCnt := _parameterCnt + 1;
  END_IF

  // Check parameter must be added ?
  IF ( CheckAddParameter(CreateCommandPayload.PayloadPtr))
  THEN
    // add command.Reserve
    CreateCommandPayload.AddByte(_command.Reserve);
    // inc parameter counter
   _parameterCnt := _parameterCnt + 1;
  END_IF

  // Check parameter must be added ?
  IF ( CheckAddParameter(CreateCommandPayload.PayloadPtr))
  THEN
    // add command.VelocityRate
    CreateCommandPayload.AddUint(_command.VelocityRate);
    // inc parameter counter
   _parameterCnt := _parameterCnt + 1;
  END_IF

  // Check parameter must be added ?
  IF ( CheckAddParameter(CreateCommandPayload.PayloadPtr))
  THEN
    // add command.AccelerationRate
    CreateCommandPayload.AddUint(_command.AccelerationRate);
    // inc parameter counter
   _parameterCnt := _parameterCnt + 1;
  END_IF

  // Check parameter must be added ?
  IF ( CheckAddParameter(CreateCommandPayload.PayloadPtr))
  THEN
    // add command.DecelerationRate
    CreateCommandPayload.AddUint(_command.DecelerationRate);
    // inc parameter counter
   _parameterCnt := _parameterCnt + 1;
  END_IF

  // Check parameter must be added ?
  IF ( CheckAddParameter(CreateCommandPayload.PayloadPtr))
  THEN
    // add command.JerkRate
    CreateCommandPayload.AddUint(_command.JerkRate);
    // inc parameter counter
   _parameterCnt := _parameterCnt + 1;
  END_IF

  // Check parameter must be added ?
  IF ( CheckAddParameter(CreateCommandPayload.PayloadPtr))
  THEN
    // add command.ToolNo
    CreateCommandPayload.AddUsint(_command.ToolNo);
    // inc parameter counter
   _parameterCnt := _parameterCnt + 1;
  END_IF

  // Check parameter must be added ?
  IF ( CheckAddParameter(CreateCommandPayload.PayloadPtr))
  THEN
    // add command.mFrameNo
    CreateCommandPayload.AddUsint(_command.FrameNo);
    // inc parameter counter
   _parameterCnt := _parameterCnt + 1;
  END_IF

  // Check parameter must be added ?
  IF ( CheckAddParameter(CreateCommandPayload.PayloadPtr))
  THEN
    // add command.BlendingMode
    CreateCommandPayload.AddUsint(_command.BlendingMode);
    // inc parameter counter
   _parameterCnt := _parameterCnt + 1;
  END_IF

  // Check parameter must be added ?
  IF ( CheckAddParameter(CreateCommandPayload.PayloadPtr))
  THEN
    // add command.OriMode
    CreateCommandPayload.AddUsint(_command.OriMode);
    // inc parameter counter
   _parameterCnt := _parameterCnt + 1;
  END_IF

  // Check parameter must be added ?
  IF ( CheckAddParameter(CreateCommandPayload.PayloadPtr))
  THEN
    // add command.BlendingParameter[0]
    CreateCommandPayload.AddReal(_command.BlendingParameter[0]);
    // inc parameter counter
   _parameterCnt := _parameterCnt + 1;
  END_IF

  // Check parameter must be added ?
  IF ( CheckAddParameter(CreateCommandPayload.PayloadPtr))
  THEN
    // add command.BlendingParameter[1]
    CreateCommandPayload.AddReal(_command.BlendingParameter[1]);
    // inc parameter counter
   _parameterCnt := _parameterCnt + 1;
  END_IF

  // Check parameter must be added ?
  IF ( CheckAddParameter(CreateCommandPayload.PayloadPtr))
  THEN
    // add command.ReferencePosition.X
    CreateCommandPayload.AddReal(_command.ReferencePosition.X);
    // inc parameter counter
   _parameterCnt := _parameterCnt + 1;
  END_IF

  // Check parameter must be added ?
  IF ( CheckAddParameter(CreateCommandPayload.PayloadPtr))
  THEN
    // add command.ReferencePosition.Y
    CreateCommandPayload.AddReal(_command.ReferencePosition.Y);
    // inc parameter counter
   _parameterCnt := _parameterCnt + 1;
  END_IF

  // Check parameter must be added ?
  IF ( CheckAddParameter(CreateCommandPayload.PayloadPtr))
  THEN
    // add command.ReferencePosition.Z
    CreateCommandPayload.AddReal(_command.ReferencePosition.Z);
    // inc parameter counter
   _parameterCnt := _parameterCnt + 1;
  END_IF

  // Check parameter must be added ?
  IF ( CheckAddParameter(CreateCommandPayload.PayloadPtr))
  THEN
    // add command.ReferencePosition.Rx
    CreateCommandPayload.AddReal(_command.ReferencePosition.Rx);
    // inc parameter counter
   _parameterCnt := _parameterCnt + 1;
  END_IF

  // Check parameter must be added ?
  IF ( CheckAddParameter(CreateCommandPayload.PayloadPtr))
  THEN
    // add command.ReferencePosition.Ry
    CreateCommandPayload.AddReal(_command.ReferencePosition.Ry);
    // inc parameter counter
   _parameterCnt := _parameterCnt + 1;
  END_IF

  // Check parameter must be added ?
  IF ( CheckAddParameter(CreateCommandPayload.PayloadPtr))
  THEN
    // add command.ReferencePosition.Rz
    CreateCommandPayload.AddReal(_command.ReferencePosition.Rz);
    // inc parameter counter
   _parameterCnt := _parameterCnt + 1;
  END_IF

  // Check parameter must be added ?
  IF ( CheckAddParameter(CreateCommandPayload.PayloadPtr))
  THEN
    // add command.ReferencePosition.Config
    CreateCommandPayload.AddArmConfig(_command.ReferencePosition.Config);
    // inc parameter counter
   _parameterCnt := _parameterCnt + 1;
  END_IF

  // Check parameter must be added ?
  IF ( CheckAddParameter(CreateCommandPayload.PayloadPtr))
  THEN
    // add command.ReferencePosition.TurnNumber
    CreateCommandPayload.AddTurnNumber(_command.ReferencePosition.TurnNumber);
    // inc parameter counter
   _parameterCnt := _parameterCnt + 1;
  END_IF

  // Check parameter must be added ?
  IF ( CheckAddParameter(CreateCommandPayload.PayloadPtr))
  THEN
    // add command.ReferencePosition.E1
    CreateCommandPayload.AddReal(_command.ReferencePosition.E1);
    // inc parameter counter
   _parameterCnt := _parameterCnt + 1;
  END_IF

  // Check parameter must be added ?
  IF ( CheckAddParameter(CreateCommandPayload.PayloadPtr))
  THEN
    // add command.Offset.X
    CreateCommandPayload.AddReal(_command.Offset.X);
    // inc parameter counter
   _parameterCnt := _parameterCnt + 1;
  END_IF

  // Check parameter must be added ?
  IF ( CheckAddParameter(CreateCommandPayload.PayloadPtr))
  THEN
    // add command.Offset.Y
    CreateCommandPayload.AddReal(_command.Offset.Y);
    // inc parameter counter
   _parameterCnt := _parameterCnt + 1;
  END_IF

  // Check parameter must be added ?
  IF ( CheckAddParameter(CreateCommandPayload.PayloadPtr))
  THEN
    // add command.Offset.Z
    CreateCommandPayload.AddReal(_command.Offset.Z);
    // inc parameter counter
   _parameterCnt := _parameterCnt + 1;
  END_IF

  // Check parameter must be added ?
  IF ( CheckAddParameter(CreateCommandPayload.PayloadPtr))
  THEN
    // add command.Offset.Rx
    CreateCommandPayload.AddReal(_command.Offset.Rx);
    // inc parameter counter
   _parameterCnt := _parameterCnt + 1;
  END_IF

  // Check parameter must be added ?
  IF ( CheckAddParameter(CreateCommandPayload.PayloadPtr))
  THEN
    // add command.Offset.Ry
    CreateCommandPayload.AddReal(_command.Offset.Ry);
    // inc parameter counter
   _parameterCnt := _parameterCnt + 1;
  END_IF

  // Check parameter must be added ?
  IF ( CheckAddParameter(CreateCommandPayload.PayloadPtr))
  THEN
    // add command.Offset.Rz
    CreateCommandPayload.AddReal(_command.Offset.Rz);
    // inc parameter counter
   _parameterCnt := _parameterCnt + 1;
  END_IF

  // Check parameter must be added ?
  IF ( CheckAddParameter(CreateCommandPayload.PayloadPtr))
  THEN
    // add command.Offset.Config
    CreateCommandPayload.AddArmConfig(_command.Offset.Config);
    // inc parameter counter
   _parameterCnt := _parameterCnt + 1;
  END_IF

  // Check parameter must be added ?
  IF ( CheckAddParameter(CreateCommandPayload.PayloadPtr))
  THEN
    // add command.Offset.TurnNumber
    CreateCommandPayload.AddTurnNumber(_command.Offset.TurnNumber);
    // inc parameter counter
   _parameterCnt := _parameterCnt + 1;
  END_IF

  // Check parameter must be added ?
  IF ( CheckAddParameter(CreateCommandPayload.PayloadPtr))
  THEN
    // add command.Offset.E1
    CreateCommandPayload.AddReal(_command.Offset.E1);
    // inc parameter counter
   _parameterCnt := _parameterCnt + 1;
  END_IF

  // Check parameter must be added ?
  IF ( CheckAddParameter(CreateCommandPayload.PayloadPtr))
  THEN
    // add command.Manipulation
    CreateCommandPayload.AddBool(_command.Manipulation);
    // inc parameter counter
   _parameterCnt := _parameterCnt + 1;
  END_IF

  // Check parameter must be added ?
  IF ( CheckAddParameter(CreateCommandPayload.PayloadPtr))
  THEN
    // add command.Reserve2
    CreateCommandPayload.AddByte(_command.Reserve2);
    // inc parameter counter
   _parameterCnt := _parameterCnt + 1;
  END_IF

  // Check parameter must be added ?
  IF ( CheckAddParameter(CreateCommandPayload.PayloadPtr))
  THEN
    // add command.ConfigMode[0]
    CreateCommandPayload.AddByte(_command.ConfigMode[0]);
    // inc parameter counter
   _parameterCnt := _parameterCnt + 1;
  END_IF

  // Check parameter must be added ?
  IF ( CheckAddParameter(CreateCommandPayload.PayloadPtr))
  THEN
    // add command.ConfigMode[1]
    CreateCommandPayload.AddByte(_command.ConfigMode[1]);
    // inc parameter counter
   _parameterCnt := _parameterCnt + 1;
  END_IF

  // Check parameter must be added ?
  IF ( CheckAddParameter(CreateCommandPayload.PayloadPtr))
  THEN
    // add command.ReferenceType
    CreateCommandPayload.AddUsint(_command.ReferenceType);
    // inc parameter counter
   _parameterCnt := _parameterCnt + 1;
  END_IF

  // Check parameter must be added ?
  IF ( CheckAddParameter(CreateCommandPayload.PayloadPtr))
  THEN
    // add command.TurnMode
    CreateCommandPayload.AddUsint(_command.TurnMode);
    // inc parameter counter
   _parameterCnt := _parameterCnt + 1;
  END_IF

  // Check parameter must be added ?
  IF ( CheckAddParameter(CreateCommandPayload.PayloadPtr))
  THEN
    // add command.MoveTime
    CreateCommandPayload.AddUint(_command.MoveTime);
    // inc parameter counter
   _parameterCnt := _parameterCnt + 1;
  END_IF

  // Check parameter must be added ?
  IF ( CheckAddParameter(CreateCommandPayload.PayloadPtr))
  THEN
    // add command.ReferencePosition.E2
    CreateCommandPayload.AddReal(_command.ReferencePosition.E2);
    // inc parameter counter
   _parameterCnt := _parameterCnt + 1;
  END_IF

  // Check parameter must be added ?
  IF ( CheckAddParameter(CreateCommandPayload.PayloadPtr))
  THEN
    // add command.ReferencePosition.E3
    CreateCommandPayload.AddReal(_command.ReferencePosition.E3);
    // inc parameter counter
   _parameterCnt := _parameterCnt + 1;
  END_IF

  // Check parameter must be added ?
  IF ( CheckAddParameter(CreateCommandPayload.PayloadPtr))
  THEN
    // add command.ReferencePosition.E4
    CreateCommandPayload.AddReal(_command.ReferencePosition.E4);
    // inc parameter counter
   _parameterCnt := _parameterCnt + 1;
  END_IF

  // Check parameter must be added ?
  IF ( CheckAddParameter(CreateCommandPayload.PayloadPtr))
  THEN
    // add command.ReferencePosition.E5
    CreateCommandPayload.AddReal(_command.ReferencePosition.E5);
    // inc parameter counter
   _parameterCnt := _parameterCnt + 1;
  END_IF

  // Check parameter must be added ?
  IF ( CheckAddParameter(CreateCommandPayload.PayloadPtr))
  THEN
    // add command.ReferencePosition.E6
    CreateCommandPayload.AddReal(_command.ReferencePosition.E6);
    // inc parameter counter
   _parameterCnt := _parameterCnt + 1;
  END_IF

  // Check parameter must be added ?
  IF ( CheckAddParameter(CreateCommandPayload.PayloadPtr))
  THEN
    // add command.Offset.E2
    CreateCommandPayload.AddReal(_command.Offset.E2);
    // inc parameter counter
   _parameterCnt := _parameterCnt + 1;
  END_IF

  // Check parameter must be added ?
  IF ( CheckAddParameter(CreateCommandPayload.PayloadPtr))
  THEN
    // add command.Offset.E3
    CreateCommandPayload.AddReal(_command.Offset.E3);
    // inc parameter counter
   _parameterCnt := _parameterCnt + 1;
  END_IF

  // Check parameter must be added ?
  IF ( CheckAddParameter(CreateCommandPayload.PayloadPtr))
  THEN
    // add command.Offset.E4
    CreateCommandPayload.AddReal(_command.Offset.E4);
    // inc parameter counter
   _parameterCnt := _parameterCnt + 1;
  END_IF

  // Check parameter must be added ?
  IF ( CheckAddParameter(CreateCommandPayload.PayloadPtr))
  THEN
    // add command.Offset.E5
    CreateCommandPayload.AddReal(_command.Offset.E5);
    // inc parameter counter
   _parameterCnt := _parameterCnt + 1;
  END_IF

  // Check parameter must be added ?
  IF ( CheckAddParameter(CreateCommandPayload.PayloadPtr))
  THEN
    // add command.Offset.E6
    CreateCommandPayload.AddReal(_command.Offset.E6);
    // inc parameter counter
   _parameterCnt := _parameterCnt + 1;
  END_IF

  // Create logging
  CreateCommandPayloadLog(AxesGroup := AxesGroup, ParameterCnt := _parameterCnt);

END_METHOD

METHOD INTERNAL CreateCommandPayloadLog
VAR_IN_OUT
  /// Robot assignment of function
  AxesGroup : AxesGroup;
END_VAR
VAR_INPUT
  /// Parameter count
  ParameterCnt : DINT;
END_VAR
VAR
  /// internal index for loops
 _idx : DINT;
END_VAR

  // Create log entry for Parameter start
  CreateLogMessagePara1 ( Timestamp   := AxesGroup.State.SystemTime,
                          MessageType := MessageType.CMD,
                          Severity    := Severity.DEBUG,
                          MessageCode := 0,
                          MessageText := 'Create command payload with the {1} parameter(s) :',
                          Para1       := DINT_TO_STRING(ParameterCnt));

  // Create log entry for EmitterID[x]
  FOR _idx := 0 TO 3
  DO
    // Return if no parameter is remaining...
    IF ( ParameterCnt = 0 ) THEN RETURN; END_IF
    // dec remaining parameter(s)
    ParameterCnt := ParameterCnt - 1;
    // Create log entry for Command.EmitterID
    CreateLogMessagePara2 ( Timestamp   := AxesGroup.State.SystemTime,
                            MessageType := MessageType.CMD,
                            Severity    := Severity.DEBUG,
                            MessageCode := 0,
                            MessageText := 'Command.EmitterID[{2}] = {1}',
                            Para1       :=  SINT_TO_STRING(_command.EmitterID[_idx]),
                            Para2       :=  DINT_TO_STRING(_idx));
  END_FOR

  // Return if no parameter is remaining...
  IF ( ParameterCnt = 0 ) THEN RETURN; END_IF
  // dec remaining parameter(s)
  ParameterCnt := ParameterCnt - 1;
  // Create log entry for ListenerID
  CreateLogMessagePara1 ( Timestamp   := AxesGroup.State.SystemTime,
                          MessageType := MessageType.CMD,
                          Severity    := Severity.DEBUG,
                          MessageCode := 0,
                          MessageText := 'Command.ListenerID = {1}',
                          Para1       :=  SINT_TO_STRING(_command.ListenerID));

  // Return if no parameter is remaining...
  IF ( ParameterCnt = 0 ) THEN RETURN; END_IF
  // dec remaining parameter(s)
  ParameterCnt := ParameterCnt - 1;
  // Create log entry for Reserve
  CreateLogMessagePara1 ( Timestamp   := AxesGroup.State.SystemTime,
                          MessageType := MessageType.CMD,
                          Severity    := Severity.DEBUG,
                          MessageCode := 0,
                          MessageText := 'Command.Reserve = {1}',
                          Para1       :=  BYTE_TO_STRING(_command.Reserve));

  // Return if no parameter is remaining...
  IF ( ParameterCnt = 0 ) THEN RETURN; END_IF
  // dec remaining parameter(s)
  ParameterCnt := ParameterCnt - 1;
  // Create log entry for VelocityRate
  CreateLogMessagePara1 ( Timestamp   := AxesGroup.State.SystemTime,
                          MessageType := MessageType.CMD,
                          Severity    := Severity.DEBUG,
                          MessageCode := 0,
                          MessageText := 'Command.VelocityRate = {1}',
                          Para1       :=  UINT_TO_STRING(_command.VelocityRate));

  // Return if no parameter is remaining...
  IF ( ParameterCnt = 0 ) THEN RETURN; END_IF
  // dec remaining parameter(s)
  ParameterCnt := ParameterCnt - 1;
  // Create log entry for AccelerationRate
  CreateLogMessagePara1 ( Timestamp   := AxesGroup.State.SystemTime,
                          MessageType := MessageType.CMD,
                          Severity    := Severity.DEBUG,
                          MessageCode := 0,
                          MessageText := 'Command.AccelerationRate = {1}',
                          Para1       :=  UINT_TO_STRING(_command.AccelerationRate));

  // Return if no parameter is remaining...
  IF ( ParameterCnt = 0 ) THEN RETURN; END_IF
  // dec remaining parameter(s)
  ParameterCnt := ParameterCnt - 1;
  // Create log entry for DecelerationRate
  CreateLogMessagePara1 ( Timestamp   := AxesGroup.State.SystemTime,
                          MessageType := MessageType.CMD,
                          Severity    := Severity.DEBUG,
                          MessageCode := 0,
                          MessageText := 'Command.DecelerationRate = {1}',
                          Para1       :=  UINT_TO_STRING(_command.DecelerationRate));

  // Return if no parameter is remaining...
  IF ( ParameterCnt = 0 ) THEN RETURN; END_IF
  // dec remaining parameter(s)
  ParameterCnt := ParameterCnt - 1;
  // Create log entry for JerkRate
  CreateLogMessagePara1 ( Timestamp   := AxesGroup.State.SystemTime,
                          MessageType := MessageType.CMD,
                          Severity    := Severity.DEBUG,
                          MessageCode := 0,
                          MessageText := 'Command.JerkRate = {1}',
                          Para1       :=  UINT_TO_STRING(_command.JerkRate));

  // Return if no parameter is remaining...
  IF ( ParameterCnt = 0 ) THEN RETURN; END_IF
  // dec remaining parameter(s)
  ParameterCnt := ParameterCnt - 1;
  // Create log entry for ToolNo
  CreateLogMessagePara1 ( Timestamp   := AxesGroup.State.SystemTime,
                          MessageType := MessageType.CMD,
                          Severity    := Severity.DEBUG,
                          MessageCode := 0,
                          MessageText := 'Command.ToolNo = {1}',
                          Para1       :=  USINT_TO_STRING(_command.ToolNo));

  // Return if no parameter is remaining...
  IF ( ParameterCnt = 0 ) THEN RETURN; END_IF
  // dec remaining parameter(s)
  ParameterCnt := ParameterCnt - 1;
  // Create log entry for FrameNo
  CreateLogMessagePara1 ( Timestamp   := AxesGroup.State.SystemTime,
                          MessageType := MessageType.CMD,
                          Severity    := Severity.DEBUG,
                          MessageCode := 0,
                          MessageText := 'Command.FrameNo = {1}',
                          Para1       :=  USINT_TO_STRING(_command.FrameNo));

  // Return if no parameter is remaining...
  IF ( ParameterCnt = 0 ) THEN RETURN; END_IF
  // dec remaining parameter(s)
  ParameterCnt := ParameterCnt - 1;
  // Create log entry for BlendingMode
  CreateLogMessagePara1 ( Timestamp   := AxesGroup.State.SystemTime,
                          MessageType := MessageType.CMD,
                          Severity    := Severity.DEBUG,
                          MessageCode := 0,
                          MessageText := 'Command.BlendingMode = {1}',
                          Para1       :=  BLENDING_MODE_TO_STRING(_command.BlendingMode));

  // Return if no parameter is remaining...
  IF ( ParameterCnt = 0 ) THEN RETURN; END_IF
  // dec remaining parameter(s)
  ParameterCnt := ParameterCnt - 1;
  // Create log entry for OriMode
  CreateLogMessagePara1 ( Timestamp   := AxesGroup.State.SystemTime,
                          MessageType := MessageType.CMD,
                          Severity    := Severity.DEBUG,
                          MessageCode := 0,
                          MessageText := 'Command.OriMode = {1}',
                          Para1       :=  ORI_MODE_TO_STRING(_command.OriMode));

  // Return if no parameter is remaining...
  IF ( ParameterCnt = 0 ) THEN RETURN; END_IF
  // dec remaining parameter(s)
  ParameterCnt := ParameterCnt - 1;
  // Create log entry for BlendingParameter[0]
  CreateLogMessagePara1 ( Timestamp   := AxesGroup.State.SystemTime,
                          MessageType := MessageType.CMD,
                          Severity    := Severity.DEBUG,
                          MessageCode := 0,
                          MessageText := 'Command.BlendingParameter[0] = {1}',
                          Para1       :=  REAL_TO_STRING(_command.BlendingParameter[0]));

  // Return if no parameter is remaining...
  IF ( ParameterCnt = 0 ) THEN RETURN; END_IF
  // dec remaining parameter(s)
  ParameterCnt := ParameterCnt - 1;
  // Create log entry for BlendingParameter[1]
  CreateLogMessagePara1 ( Timestamp   := AxesGroup.State.SystemTime,
                          MessageType := MessageType.CMD,
                          Severity    := Severity.DEBUG,
                          MessageCode := 0,
                          MessageText := 'Command.BlendingParameter[1] = {1}',
                          Para1       :=  REAL_TO_STRING(_command.BlendingParameter[1]));

  // Return if no parameter is remaining...
  IF ( ParameterCnt = 0 ) THEN RETURN; END_IF
  // dec remaining parameter(s)
  ParameterCnt := ParameterCnt - 1;
  // Create log entry for ReferencePosition.X
  CreateLogMessagePara1 ( Timestamp   := AxesGroup.State.SystemTime,
                          MessageType := MessageType.CMD,
                          Severity    := Severity.DEBUG,
                          MessageCode := 0,
                          MessageText := 'Command.ReferencePosition.X = {1}',
                          Para1       :=  REAL_TO_STRING(_command.ReferencePosition.X));

  // Return if no parameter is remaining...
  IF ( ParameterCnt = 0 ) THEN RETURN; END_IF
  // dec remaining parameter(s)
  ParameterCnt := ParameterCnt - 1;
  // Create log entry for ReferencePosition.Y
  CreateLogMessagePara1 ( Timestamp   := AxesGroup.State.SystemTime,
                          MessageType := MessageType.CMD,
                          Severity    := Severity.DEBUG,
                          MessageCode := 0,
                          MessageText := 'Command.ReferencePosition.Y = {1}',
                          Para1       :=  REAL_TO_STRING(_command.ReferencePosition.Y));

  // Return if no parameter is remaining...
  IF ( ParameterCnt = 0 ) THEN RETURN; END_IF
  // dec remaining parameter(s)
  ParameterCnt := ParameterCnt - 1;
  // Create log entry for ReferencePosition.Z
  CreateLogMessagePara1 ( Timestamp   := AxesGroup.State.SystemTime,
                          MessageType := MessageType.CMD,
                          Severity    := Severity.DEBUG,
                          MessageCode := 0,
                          MessageText := 'Command.ReferencePosition.Z = {1}',
                          Para1       :=  REAL_TO_STRING(_command.ReferencePosition.Z));

  // Return if no parameter is remaining...
  IF ( ParameterCnt = 0 ) THEN RETURN; END_IF
  // dec remaining parameter(s)
  ParameterCnt := ParameterCnt - 1;
  // Create log entry for ReferencePosition.Rx
  CreateLogMessagePara1 ( Timestamp   := AxesGroup.State.SystemTime,
                          MessageType := MessageType.CMD,
                          Severity    := Severity.DEBUG,
                          MessageCode := 0,
                          MessageText := 'Command.ReferencePosition.Rx = {1}',
                          Para1       :=  REAL_TO_STRING(_command.ReferencePosition.Rx));

  // Return if no parameter is remaining...
  IF ( ParameterCnt = 0 ) THEN RETURN; END_IF
  // dec remaining parameter(s)
  ParameterCnt := ParameterCnt - 1;
  // Create log entry for ReferencePosition.Ry
  CreateLogMessagePara1 ( Timestamp   := AxesGroup.State.SystemTime,
                          MessageType := MessageType.CMD,
                          Severity    := Severity.DEBUG,
                          MessageCode := 0,
                          MessageText := 'Command.ReferencePosition.Ry = {1}',
                          Para1       :=  REAL_TO_STRING(_command.ReferencePosition.Ry));

  // Return if no parameter is remaining...
  IF ( ParameterCnt = 0 ) THEN RETURN; END_IF
  // dec remaining parameter(s)
  ParameterCnt := ParameterCnt - 1;
  // Create log entry for ReferencePosition.Rz
  CreateLogMessagePara1 ( Timestamp   := AxesGroup.State.SystemTime,
                          MessageType := MessageType.CMD,
                          Severity    := Severity.DEBUG,
                          MessageCode := 0,
                          MessageText := 'Command.ReferencePosition.Rz = {1}',
                          Para1       :=  REAL_TO_STRING(_command.ReferencePosition.Rz));

  // Return if no parameter is remaining...
  IF ( ParameterCnt = 0 ) THEN RETURN; END_IF
  // dec remaining parameter(s)
  ParameterCnt := ParameterCnt - 1;
  // Create log entry for ReferencePosition.Config
  CreateLogMessagePara1 ( Timestamp   := AxesGroup.State.SystemTime,
                          MessageType := MessageType.CMD,
                          Severity    := Severity.DEBUG,
                          MessageCode := 0,
                          MessageText := 'Command.ReferencePosition.Config = {1}',
                          Para1       :=  ARM_CONFIG_TO_STRING(_command.ReferencePosition.Config));

  // Return if no parameter is remaining...
  IF ( ParameterCnt = 0 ) THEN RETURN; END_IF
  // dec remaining parameter(s)
  ParameterCnt := ParameterCnt - 1;
  // Create log entry for ReferencePosition.Reserve
  CreateLogMessagePara1 ( Timestamp   := AxesGroup.State.SystemTime,
                          MessageType := MessageType.CMD,
                          Severity    := Severity.DEBUG,
                          MessageCode := 0,
                          MessageText := 'Command.ReferencePosition.Reserve = {1}',
                          Para1       :=  BYTE_TO_STRING(0));

  // Return if no parameter is remaining...
  IF ( ParameterCnt = 0 ) THEN RETURN; END_IF
  // dec remaining parameter(s)
  ParameterCnt := ParameterCnt - 1;
  // Create log entry for ReferencePosition.TurnNumber[0]
  CreateLogMessagePara1 ( Timestamp   := AxesGroup.State.SystemTime,
                          MessageType := MessageType.CMD,
                          Severity    := Severity.DEBUG,
                          MessageCode := 0,
                          MessageText := 'Command.ReferencePosition.TurnNumber[0] = {1}',
                          Para1       :=  BYTE_TO_STRING(CombineHalfSints(HalfSintHi := _command.ReferencePosition.TurnNumber.J2Turns,
                                                                          HalfSintLo := _command.ReferencePosition.TurnNumber.J1Turns)));

  // Return if no parameter is remaining...
  IF ( ParameterCnt = 0 ) THEN RETURN; END_IF
  // dec remaining parameter(s)
  ParameterCnt := ParameterCnt - 1;
  // Create log entry for ReferencePosition.TurnNumber[1]
  CreateLogMessagePara1 ( Timestamp   := AxesGroup.State.SystemTime,
                          MessageType := MessageType.CMD,
                          Severity    := Severity.DEBUG,
                          MessageCode := 0,
                          MessageText := 'Command.ReferencePosition.TurnNumber[1] = {1}',
                          Para1       :=  BYTE_TO_STRING(CombineHalfSints(HalfSintHi := _command.ReferencePosition.TurnNumber.J4Turns,
                                                                          HalfSintLo := _command.ReferencePosition.TurnNumber.J3Turns)));

  // Return if no parameter is remaining...
  IF ( ParameterCnt = 0 ) THEN RETURN; END_IF
  // dec remaining parameter(s)
  ParameterCnt := ParameterCnt - 1;
  // Create log entry for ReferencePosition.TurnNumber[2]
  CreateLogMessagePara1 ( Timestamp   := AxesGroup.State.SystemTime,
                          MessageType := MessageType.CMD,
                          Severity    := Severity.DEBUG,
                          MessageCode := 0,
                          MessageText := 'Command.ReferencePosition.TurnNumber[2] = {1}',
                          Para1       :=  BYTE_TO_STRING(CombineHalfSints(HalfSintHi := _command.ReferencePosition.TurnNumber.J6Turns,
                                                                          HalfSintLo := _command.ReferencePosition.TurnNumber.J5Turns)));

  // Return if no parameter is remaining...
  IF ( ParameterCnt = 0 ) THEN RETURN; END_IF
  // dec remaining parameter(s)
  ParameterCnt := ParameterCnt - 1;
  // Create log entry for ReferencePosition.TurnNumber[3]
  CreateLogMessagePara1 ( Timestamp   := AxesGroup.State.SystemTime,
                          MessageType := MessageType.CMD,
                          Severity    := Severity.DEBUG,
                          MessageCode := 0,
                          MessageText := 'Command.ReferencePosition.TurnNumber[3] = {1}',
                          Para1       :=  SINT_TO_STRING(_command.ReferencePosition.TurnNumber.E1Turns));

  // Return if no parameter is remaining...
  IF ( ParameterCnt = 0 ) THEN RETURN; END_IF
  // dec remaining parameter(s)
  ParameterCnt := ParameterCnt - 1;
  // Create log entry for ReferencePosition.E1
  CreateLogMessagePara1 ( Timestamp   := AxesGroup.State.SystemTime,
                          MessageType := MessageType.CMD,
                          Severity    := Severity.DEBUG,
                          MessageCode := 0,
                          MessageText := 'Command.ReferencePosition.E1 = {1}',
                          Para1       :=  REAL_TO_STRING(_command.ReferencePosition.E1));

  // Return if no parameter is remaining...
  IF ( ParameterCnt = 0 ) THEN RETURN; END_IF
  // dec remaining parameter(s)
  ParameterCnt := ParameterCnt - 1;
  // Create log entry for Offset.X
  CreateLogMessagePara1 ( Timestamp   := AxesGroup.State.SystemTime,
                          MessageType := MessageType.CMD,
                          Severity    := Severity.DEBUG,
                          MessageCode := 0,
                          MessageText := 'Command.Offset.X = {1}',
                          Para1       :=  REAL_TO_STRING(_command.Offset.X));

  // Return if no parameter is remaining...
  IF ( ParameterCnt = 0 ) THEN RETURN; END_IF
  // dec remaining parameter(s)
  ParameterCnt := ParameterCnt - 1;
  // Create log entry for Offset.Y
  CreateLogMessagePara1 ( Timestamp   := AxesGroup.State.SystemTime,
                          MessageType := MessageType.CMD,
                          Severity    := Severity.DEBUG,
                          MessageCode := 0,
                          MessageText := 'Command.Offset.Y = {1}',
                          Para1       :=  REAL_TO_STRING(_command.Offset.Y));

  // Return if no parameter is remaining...
  IF ( ParameterCnt = 0 ) THEN RETURN; END_IF
  // dec remaining parameter(s)
  ParameterCnt := ParameterCnt - 1;
  // Create log entry for Offset.Z
  CreateLogMessagePara1 ( Timestamp   := AxesGroup.State.SystemTime,
                          MessageType := MessageType.CMD,
                          Severity    := Severity.DEBUG,
                          MessageCode := 0,
                          MessageText := 'Command.Offset.Z = {1}',
                          Para1       :=  REAL_TO_STRING(_command.Offset.Z));

  // Return if no parameter is remaining...
  IF ( ParameterCnt = 0 ) THEN RETURN; END_IF
  // dec remaining parameter(s)
  ParameterCnt := ParameterCnt - 1;
  // Create log entry for Offset.Rx
  CreateLogMessagePara1 ( Timestamp   := AxesGroup.State.SystemTime,
                          MessageType := MessageType.CMD,
                          Severity    := Severity.DEBUG,
                          MessageCode := 0,
                          MessageText := 'Command.Offset.Rx = {1}',
                          Para1       :=  REAL_TO_STRING(_command.Offset.Rx));

  // Return if no parameter is remaining...
  IF ( ParameterCnt = 0 ) THEN RETURN; END_IF
  // dec remaining parameter(s)
  ParameterCnt := ParameterCnt - 1;
  // Create log entry for Offset.Ry
  CreateLogMessagePara1 ( Timestamp   := AxesGroup.State.SystemTime,
                          MessageType := MessageType.CMD,
                          Severity    := Severity.DEBUG,
                          MessageCode := 0,
                          MessageText := 'Command.Offset.Ry = {1}',
                          Para1       :=  REAL_TO_STRING(_command.Offset.Ry));

  // Return if no parameter is remaining...
  IF ( ParameterCnt = 0 ) THEN RETURN; END_IF
  // dec remaining parameter(s)
  ParameterCnt := ParameterCnt - 1;
  // Create log entry for Offset.Rz
  CreateLogMessagePara1 ( Timestamp   := AxesGroup.State.SystemTime,
                          MessageType := MessageType.CMD,
                          Severity    := Severity.DEBUG,
                          MessageCode := 0,
                          MessageText := 'Command.Offset.Rz = {1}',
                          Para1       :=  REAL_TO_STRING(_command.Offset.Rz));

  // Return if no parameter is remaining...
  IF ( ParameterCnt = 0 ) THEN RETURN; END_IF
  // dec remaining parameter(s)
  ParameterCnt := ParameterCnt - 1;
  // Create log entry for Offset.Config
  CreateLogMessagePara1 ( Timestamp   := AxesGroup.State.SystemTime,
                          MessageType := MessageType.CMD,
                          Severity    := Severity.DEBUG,
                          MessageCode := 0,
                          MessageText := 'Command.Offset.Config = {1}',
                          Para1       :=  ARM_CONFIG_TO_STRING(_command.Offset.Config));

  // Return if no parameter is remaining...
  IF ( ParameterCnt = 0 ) THEN RETURN; END_IF
  // dec remaining parameter(s)
  ParameterCnt := ParameterCnt - 1;
  // Create log entry for Offset.Reserve
  CreateLogMessagePara1 ( Timestamp   := AxesGroup.State.SystemTime,
                          MessageType := MessageType.CMD,
                          Severity    := Severity.DEBUG,
                          MessageCode := 0,
                          MessageText := 'Command.Offset.Reserve = {1}',
                          Para1       :=  BYTE_TO_STRING(0));

  // Return if no parameter is remaining...
  IF ( ParameterCnt = 0 ) THEN RETURN; END_IF
  // dec remaining parameter(s)
  ParameterCnt := ParameterCnt - 1;
  // Create log entry for Offset.TurnNumber[0]
  CreateLogMessagePara1 ( Timestamp   := AxesGroup.State.SystemTime,
                          MessageType := MessageType.CMD,
                          Severity    := Severity.DEBUG,
                          MessageCode := 0,
                          MessageText := 'Command.Offset.TurnNumber[0] = {1}',
                          Para1       :=  BYTE_TO_STRING(CombineHalfSints(HalfSintHi := _command.Offset.TurnNumber.J2Turns,
                                                                          HalfSintLo := _command.Offset.TurnNumber.J1Turns)));

  // Return if no parameter is remaining...
  IF ( ParameterCnt = 0 ) THEN RETURN; END_IF
  // dec remaining parameter(s)
  ParameterCnt := ParameterCnt - 1;
  // Create log entry for Offset.TurnNumber[1]
  CreateLogMessagePara1 ( Timestamp   := AxesGroup.State.SystemTime,
                          MessageType := MessageType.CMD,
                          Severity    := Severity.DEBUG,
                          MessageCode := 0,
                          MessageText := 'Command.Offset.TurnNumber[1] = {1}',
                          Para1       :=  BYTE_TO_STRING(CombineHalfSints(HalfSintHi := _command.Offset.TurnNumber.J4Turns,
                                                                          HalfSintLo := _command.Offset.TurnNumber.J3Turns)));

  // Return if no parameter is remaining...
  IF ( ParameterCnt = 0 ) THEN RETURN; END_IF
  // dec remaining parameter(s)
  ParameterCnt := ParameterCnt - 1;
  // Create log entry for Offset.TurnNumber[2]
  CreateLogMessagePara1 ( Timestamp   := AxesGroup.State.SystemTime,
                          MessageType := MessageType.CMD,
                          Severity    := Severity.DEBUG,
                          MessageCode := 0,
                          MessageText := 'Command.Offset.TurnNumber[2] = {1}',
                          Para1       :=  BYTE_TO_STRING(CombineHalfSints(HalfSintHi := _command.Offset.TurnNumber.J6Turns,
                                                                          HalfSintLo := _command.Offset.TurnNumber.J5Turns)));

  // Return if no parameter is remaining...
  IF ( ParameterCnt = 0 ) THEN RETURN; END_IF
  // dec remaining parameter(s)
  ParameterCnt := ParameterCnt - 1;
  // Create log entry for Offset.TurnNumber[3]
  CreateLogMessagePara1 ( Timestamp   := AxesGroup.State.SystemTime,
                          MessageType := MessageType.CMD,
                          Severity    := Severity.DEBUG,
                          MessageCode := 0,
                          MessageText := 'Command.Offset.TurnNumber[3] = {1}',
                          Para1       :=  SINT_TO_STRING(_command.Offset.TurnNumber.E1Turns));

  // Return if no parameter is remaining...
  IF ( ParameterCnt = 0 ) THEN RETURN; END_IF
  // dec remaining parameter(s)
  ParameterCnt := ParameterCnt - 1;
  // Create log entry for Offset.E1
  CreateLogMessagePara1 ( Timestamp   := AxesGroup.State.SystemTime,
                          MessageType := MessageType.CMD,
                          Severity    := Severity.DEBUG,
                          MessageCode := 0,
                          MessageText := 'Command.Offset.E1 = {1}',
                          Para1       :=  REAL_TO_STRING(_command.Offset.E1));

  // Return if no parameter is remaining...
  IF ( ParameterCnt = 0 ) THEN RETURN; END_IF
  // dec remaining parameter(s)
  ParameterCnt := ParameterCnt - 1;
  // Create log entry for Manipulation
  CreateLogMessagePara1 ( Timestamp   := AxesGroup.State.SystemTime,
                          MessageType := MessageType.CMD,
                          Severity    := Severity.DEBUG,
                          MessageCode := 0,
                          MessageText := 'Command.Manipulation = {1}',
                          Para1       :=  BOOL_TO_STRING(_command.Manipulation));

  // Return if no parameter is remaining...
  IF ( ParameterCnt = 0 ) THEN RETURN; END_IF
  // dec remaining parameter(s)
  ParameterCnt := ParameterCnt - 1;
  // Create log entry for Reserve
  CreateLogMessagePara1 ( Timestamp   := AxesGroup.State.SystemTime,
                          MessageType := MessageType.CMD,
                          Severity    := Severity.DEBUG,
                          MessageCode := 0,
                          MessageText := 'Command.Reserve = {1}',
                          Para1       :=  BYTE_TO_STRING(_command.Reserve));

  // Return if no parameter is remaining...
  IF ( ParameterCnt = 0 ) THEN RETURN; END_IF
  // dec remaining parameter(s)
  ParameterCnt := ParameterCnt - 1;
  // Create log entry for ConfigMode[0]
  CreateLogMessagePara1 ( Timestamp   := AxesGroup.State.SystemTime,
                          MessageType := MessageType.CMD,
                          Severity    := Severity.DEBUG,
                          MessageCode := 0,
                          MessageText := 'Command.ConfigMode[0] = {1}',
                          Para1       :=  BYTE_TO_STRING_BIN(_command.ConfigMode[0]));

  // Return if no parameter is remaining...
  IF ( ParameterCnt = 0 ) THEN RETURN; END_IF
  // dec remaining parameter(s)
  ParameterCnt := ParameterCnt - 1;
  // Create log entry for ConfigMode[1]
  CreateLogMessagePara1 ( Timestamp   := AxesGroup.State.SystemTime,
                          MessageType := MessageType.CMD,
                          Severity    := Severity.DEBUG,
                          MessageCode := 0,
                          MessageText := 'Command.ConfigMode[1] = {1}',
                          Para1       :=  BYTE_TO_STRING_BIN(_command.ConfigMode[1]));

  // Return if no parameter is remaining...
  IF ( ParameterCnt = 0 ) THEN RETURN; END_IF
  // dec remaining parameter(s)
  ParameterCnt := ParameterCnt - 1;
  // Create log entry for ReferenceType
  CreateLogMessagePara1 ( Timestamp   := AxesGroup.State.SystemTime,
                          MessageType := MessageType.CMD,
                          Severity    := Severity.DEBUG,
                          MessageCode := 0,
                          MessageText := 'Command.ReferenceType = {1}',
                          Para1       :=  REFERENCE_TYPE_TO_STRING(_command.ReferenceType));

  // Return if no parameter is remaining...
  IF ( ParameterCnt = 0 ) THEN RETURN; END_IF
  // dec remaining parameter(s)
  ParameterCnt := ParameterCnt - 1;
  // Create log entry for TurnMode
  CreateLogMessagePara1 ( Timestamp   := AxesGroup.State.SystemTime,
                          MessageType := MessageType.CMD,
                          Severity    := Severity.DEBUG,
                          MessageCode := 0,
                          MessageText := 'Command.TurnMode = {1}',
                          Para1       :=  TURN_MODE_TO_STRING(_command.TurnMode));
